(* Status Word *)
	stStatusData.bEnableOutputStage		:= fVelocity <> 0;
	stStatusData.bInverterReady   		:= TRUE;
	stStatusData.bPoDataEnable    		:= FALSE;
	stStatusData.bReserved3       		:= FALSE;
	stStatusData.bReserved4       		:= FALSE;
	stStatusData.bError           		:= FALSE;
	stStatusData.bReserved6       		:= FALSE;
	stStatusData.bReserved7       		:= FALSE;
	stStatusData.nStatus				:= 0;
END_METHOD

METHOD INTERNAL GetControlData
VAR_INPUT
	stControl 		: REFERENCE TO ST_SimMovitracControlData;
	pAddr			: ULINT; //PO adress
	bSwap 			: BOOL; //Swap BE_TO_HOST
END_VAR

VAR
	nCtrlIndex		: DWORD;
	nSpeedIndex		: DWORD;
	nRampIndex		: DWORD;
END_VAR
IF pAddr <= 0 THEN RETURN; END_IF

nCtrlIndex := stConfig.nCtrlAssign;
nSpeedIndex := stConfig.nSpeedAssign;
nRampIndex := stConfig.nRampAssign;

IF stConfig.bSwapProcessData THEN
	MEMCPY(ADR(stControlData) + 1, pAddr + nCtrlIndex, 1);
	MEMCPY(ADR(stControlData), pAddr + nCtrlIndex + 1, 1);
	MEMCPY(ADR(stControlData.nSetpointSpeed) + 1, pAddr + nSpeedIndex, 1);
	MEMCPY(ADR(stControlData.nSetpointSpeed), pAddr + nSpeedIndex + 1, 1);
ELSE
	MEMCPY(ADR(stControlData), pAddr + nCtrlIndex, 2);
	MEMCPY(ADR(stControlData.nSetpointSpeed), pAddr + nSpeedIndex, 2);
END_IF
END_METHOD

METHOD INTERNAL InitRun : BOOL
VAR_INST
	bInitRun : BOOL := TRUE;
END_VAR
IF NOT bInitRun THEN RETURN; END_IF
bInitRun := FALSE;

IF pControlData = 0 OR pStatusData = 0 THEN
	ADSLOGSTR(ADSLOG_MSGTYPE_WARN, CONCAT(sPath, ': %s'), 'Plc address not set.');
END_IF
END_METHOD

METHOD INTERNAL SetStatusData
VAR_INPUT
	stStatus 		: ST_SimMovitracStatusData;
	pAddr			: ULINT;
	bSwap 			: BOOL;
END_VAR

VAR
	nStatusIndex	: DWORD;
	nSpeedIndex	: DWORD;
END_VAR
IF pAddr <= 0 THEN RETURN; END_IF

nStatusIndex := stConfig.nStatusAssign;
nSpeedIndex := stConfig.nSpeedActAssign;

IF stConfig.bSwapProcessData THEN
	MEMCPY(pAddr + nStatusIndex + 1, ADR(stStatusData), 1);
	MEMCPY(pAddr + nStatusIndex, ADR(stStatusData.nStatus), 1);
	MEMCPY(pAddr + nSpeedIndex + 1, ADR(stStatusData.nActSpeed), 1);
	MEMCPY(pAddr + nSpeedIndex, ADR(stStatusData.nActSpeed) + 1, 1);	
ELSE
	MEMCPY(pAddr + nStatusIndex, ADR(stStatusData), 2);
	MEMCPY(pAddr + nSpeedIndex, ADR(stStatusData.nActSpeed), 2);
END_IF
END_METHOD

END_FUNCTION_BLOCK

// Devices/Drives/FB_SimMovitrac/FB_SimMovitracLTEB
FUNCTION_BLOCK FB_SimMovitracLTEB EXTENDS FB_LinkDataReal
VAR_INPUT
	bSTO					: BOOL := TRUE;
	bEnable 				: BOOL;
	bReverse				: BOOL;
	nTargetSpeed			: UINT; // Unit [INC]
	stConfig				: ST_SimMovitracConfig;
END_VAR

VAR_OUTPUT
	fActualSpeed			: REAL; // Units [RPM]
	bReady 					: BOOL;
	bRunning 				: BOOL;
END_VAR

VAR
	fAcc 					: REAL;
END_VAR

VAR CONSTANT
	
	MAX_VALUE_UINT 			: UINT := 65535; 
END_VAR

SUPER^();
InitRun();
ControlLogic();

METHOD PRIVATE ControlLogic
VAR
	fTargetSpeedInPercent	: REAL;
	fTargetSpeed 			: REAL;
END_VAR
// Start inverter 
IF bEnable AND bSTO THEN
	fTargetSpeedInPercent := F_Norm(0, MAX_VALUE_UINT, ABS(UINT_TO_REAL(nTargetSpeed))); // [INC] to [%] 
	fTargetSpeed := stConfig.fReferenceVelocity * fTargetSpeedInPercent; // [RPM]
	
	IF bReverse THEN
		ControlData := fTargetSpeed * -1;
	ELSE 
		ControlData := fTargetSpeed;
	END_IF
ELSE 
	ControlData := 0; 
END_IF

// Send values to the simulation interface
Control.0 := bEnable AND bSTO;

// Receive values from the simulation interface 
fActualSpeed := StatusData * stConfig.fGearFactor;
bReady  	 := NOT bEnable AND bSTO;
bRunning 	 := Status.0;
END_METHOD

METHOD PRIVATE InitRun
VAR_INST
	bInitRun : BOOL := TRUE;
END_VAR
IF NOT bInitRun THEN RETURN; END_IF
bInitRun := FALSE;

fAcc := stConfig.fReferenceVelocity * 1000 / stConfig.fProcessRamp;
END_METHOD

END_FUNCTION_BLOCK

// Devices/Drives/FB_Starter/FB_Starter
{attribute 'reflection'}
FUNCTION_BLOCK FB_Starter EXTENDS FB_LinkDataREAL
VAR_INPUT
	stControlData		: ST_StarterControlData;
	stConfig			: ST_StarterConfig;	
END_VAR

VAR_OUTPUT
	stStatusData		: ST_StarterStatusData;	
	fSpeed				: REAL; // Units [RPM]
END_VAR

VAR
	{attribute 'instance-path'}
	{attribute 'noinit'}
	sPath				: STRING;	
                    	
	fbDriveControl		: FB_DriveControl;
	bMoveActive			: BOOL;
	
	pControlData		: POINTER TO BYTE; //Addr. Process Output (PO), 2 BYTES FROM FIELDBUS
	pStatusData			: POINTER TO BYTE; //Addr. Process Input (PI), 2 BYTES FROM FIELDBUS
END_VAR

SUPER^();
InitRun();

GetControlData(stControlData, pControlData, stConfig.bSwapProcessData);
ControlLogic();
SetStatusData(stStatusData, pStatusData, stConfig.bSwapProcessData);

(*Assign Process Data Objects to device*)
METHOD PUBLIC AssignProcessData : BOOL
VAR_INPUT
	aControlData 		: ANY; //Addr. Process Output (PO), 2 BYTES FROM FIELDBUS
	aStatusData 		: ANY; //Addr. Process Input (PI), 2 BYTES TO FIELDBUS
END_VAR
THIS^.pControlData := aControlData.pValue;
THIS^.pStatusData := aStatusData.pValue;
END_METHOD

METHOD INTERNAL ControlLogic
(* Set parameter *)	
	bMoveActive := FALSE;
	
	IF (stControlData.MotorCW AND NOT stControlData.MotorCCW AND stControlData.BrakeActuation AND NOT stStatusData.GroupFault) THEN
		fbDriveControl.MoveVelocity(
			(stConfig.fVelocity),
			(stConfig.fAcceleration),
			(stConfig.fDeceleration));
		bMoveActive := TRUE;
	END_IF
	
	IF (stControlData.MotorCCW AND NOT stControlData.MotorCW AND stControlData.BrakeActuation AND NOT stStatusData.GroupFault) THEN
		fbDriveControl.MoveVelocity(
			(-stConfig.fVelocity),
			(stConfig.fAcceleration),
			(stConfig.fDeceleration));
		bMoveActive := TRUE;
	END_IF
	
	IF NOT bMoveActive OR stStatusData.GroupFault THEN
		fbDriveControl.Stop(stConfig.fDeceleration);
	END_IF

ControlData := fSpeed := fbDriveControl.fVelocity;
	
stStatusData.Ready 				:= TRUE;
stStatusData.MotorON 			:= NOT F_Compare(fbDriveControl.fVelocity, 0, 0.001); 
stStatusData.GroupFault 		:= FALSE;
stStatusData.GroupWarn 			:= FALSE;
stStatusData.Input1 			:= FALSE;
stStatusData.Input2 			:= FALSE;
stStatusData.Input3 			:= FALSE;
stStatusData.Input4 			:= FALSE;
stStatusData.MotorCurrent0 		:= FALSE;
stStatusData.MotorCurrent1 		:= FALSE;
stStatusData.MotorCurrent2 		:= FALSE;
stStatusData.MotorCurrent3 		:= FALSE;
stStatusData.MotorCurrent4 		:= FALSE;
stStatusData.MotorCurrent5 		:= FALSE;
stStatusData.ManualLocalMode	:= FALSE;
stStatusData.RampOperation 		:= FALSE;
END_METHOD

METHOD INTERNAL GetControlData
VAR_INPUT
	stControl 		: REFERENCE TO ST_StarterControlData;
	pAddr			: ULINT; //PO adress
	bSwap 			: BOOL; //Swap BE_TO_HOST
END_VAR

VAR	
	nControlWord 	: WORD;
END_VAR
IF pAddr <= 0 THEN RETURN; END_IF

IF bSwap THEN 
	MEMCPY(ADR(nControlWord), pAddr, 2);
	nControlWord := BE16_TO_HOST(nControlWord);
	MEMCPY(ADR(stControl), ADR(nControlWord), 2);
ELSE
	MEMCPY(ADR(stControl), pAddr, 2);
END_IF
END_METHOD

METHOD INTERNAL InitRun
VAR_INST
	bInitRun : BOOL := TRUE;
END_VAR
IF NOT bInitRun THEN RETURN; END_IF
bInitRun := FALSE;

IF pControlData = 0 OR pStatusData = 0 THEN
	ADSLOGSTR(ADSLOG_MSGTYPE_WARN, CONCAT(sPath, ': %s'), 'Plc address not set.');
END_IF

fbDriveControl.fPositionLimitMin := 0;
fbDriveControl.fPositionLimitMax := 0;
fbDriveControl.fAccMax := 0;
fbDriveControl.fTolerance := 0.1;
END_METHOD

METHOD INTERNAL SetStatusData
VAR_INPUT
	stStatus 		: ST_StarterStatusData;
	pAddr			: ULINT;
	bSwap 			: BOOL;
END_VAR

VAR
	nStatusWord 	: WORD;
END_VAR
IF pAddr <= 0 THEN RETURN; END_IF

IF bSwap THEN 
	MEMCPY(ADR(nStatusWord), ADR(stStatus), 2);
	nStatusWord := HOST_TO_BE16(nStatusWord);
	MEMCPY(pAddr, ADR(nStatusWord), 2);
ELSE
	MEMCPY(pAddr, ADR(stStatus), 2);
END_IF
END_METHOD

END_FUNCTION_BLOCK

// Devices/Safety/FB_EuchnerMGB
FUNCTION_BLOCK FB_EuchnerMGB EXTENDS FB_LinkDevice
VAR_INPUT
	bLock 					: BOOL; //Deactivates the tightening magnet
	bLockGuardMonitoring	: BOOL := TRUE; //Guard lock monitoring 0- 
	bReset 					: BOOL; //Error acknowledgement
	bLamp_1					: BOOL; //User defined input for item 1
	bLamp_2					: BOOL; //User defined input for item 2
	bLamp_3					: BOOL; //User defined input for item 3
	bLamp_4					: BOOL; //User defined input for item 4
END_VAR
VAR_OUTPUT
	bClosed 				: BOOL; //Door is closed
	bClosedAndLocked 		: BOOL; //Door is closed and guard locked / interlocked
	bButton_1				: BOOL; //User defined output for item 1
	bButton_2				: BOOL;	//User defined output for item 2
	bButton_3				: BOOL; //User defined output for item 3
	bButton_4				: BOOL; //User defined output for item 4
END_VAR

SUPER^();

Control.0 			:= bLock;
Control.1 			:= bReset;
Control.4 			:= bLamp_1;
Control.5 			:= bLamp_2;
Control.6 			:= bLamp_3;
Control.7 			:= bLamp_4;

bClosed 			:= Status.0;

IF bLockGuardMonitoring THEN
	bClosedAndLocked 	:= Status.1;
ELSE
	bClosedAndLocked 	:= Status.0;	
END_IF

bButton_1 			:= Status.4;
bButton_2 			:= Status.5;
bButton_3 			:= Status.6;
bButton_4 			:= Status.7;

END_FUNCTION_BLOCK

// Devices/Safety/FB_EuchnerSTP
FUNCTION_BLOCK FB_EuchnerSTP EXTENDS FB_LinkDevice
VAR_INPUT
	bLock 				: BOOL; //Deactivates the tightening magnet
	bLamp_RD			: BOOL; //User defined input for item 1
	bLamp_GN			: BOOL; //User defined input for item 2
END_VAR
VAR_OUTPUT
	bClosed 			: BOOL; //Door is closed
	bClosedAndLocked 	: BOOL; //Door is closed and guard locked / interlocked
END_VAR

SUPER^();
Control.0 			:= bLock;

Control.4 			:= bLamp_RD;
Control.5 			:= bLamp_GN;

bClosed 			:= Status.0;
bClosedAndLocked    := Status.1 OR (bLock AND bClosed);

END_FUNCTION_BLOCK

// Tests/Common/FB_AdsMessageHandler_Test
FUNCTION_BLOCK FB_AdsMessageHandler_Test EXTENDS TcUnit.FB_TestSuite
VAR
	stAdsMessageSend 		: ST_AdsMessage;
END_VAR

stAdsMessageSend.nIdxGrp := 16#80000005;
stAdsMessageSend.nIdxOffs := 7;
TestCaseWrite('ADS Write Indication 1', stAdsMessageSend);

stAdsMessageSend.nIdxGrp := 16#80000006;
stAdsMessageSend.nIdxOffs := 8;
TestCaseWrite('ADS Write Indication 2', stAdsMessageSend);

stAdsMessageSend.nIdxGrp := 16#80000007;
stAdsMessageSend.nIdxOffs := 9;
TestCaseWrite('ADS Write Indication 3', stAdsMessageSend);

stAdsMessageSend.nIdxGrp := 16#80000005;
stAdsMessageSend.nIdxOffs := 7;
TestCaseRead('ADS Read Indication 1', stAdsMessageSend);

stAdsMessageSend.nIdxGrp := 16#80000006;
stAdsMessageSend.nIdxOffs := 8;
TestCaseRead('ADS Read Indication 2', stAdsMessageSend);

stAdsMessageSend.nIdxGrp := 16#80000007;
stAdsMessageSend.nIdxOffs := 9;
TestCaseRead('ADS Read Indication 3', stAdsMessageSend);

METHOD TestCaseRead : REFERENCE TO FB_Test
VAR_INPUT
	sName 					: T_MaxString;
	stAdsMessage 			: ST_AdsMessage;
END_VAR

VAR
	fbAdsMessageHandler 	: FB_AdsMessageHandler;		
	fbAdsRead				: ADSREAD := (NETID := '', PORT := 851, TMOUT := DEFAULT_ADS_TIMEOUT);
	aData 					: ARRAY[0..5] OF BYTE;
	bResult 				: BOOL; 	
	stAdsMessageResult 	: ST_AdsMessage;
END_VAR
TEST(sName);

fbAdsRead(READ := FALSE);
fbAdsRead(IDXGRP := stAdsMessageSend.nIdxGrp, 
		IDXOFFS := stAdsMessageSend.nIdxOffs, 
        LEN := stAdsMessageSend.nLength, 
		DESTADDR := ADR(aData), 
        READ := TRUE);			

fbAdsMessageHandler.bVerbose := TRUE;			
fbAdsMessageHandler();

bResult := fbAdsMessageHandler.bIsAdsMessageReadValid;
stAdsMessageResult := fbAdsMessageHandler.stAdsMessageRead;

AssertTrue(bResult, 'Result value is not correct');

AssertEquals(Expected := stAdsMessage.tNetID,
Actual := stAdsMessageResult.tNetID,
Message := 'tNetID is not valid');

AssertEquals(Expected := stAdsMessage.nIdxGrp,
Actual := stAdsMessageResult.nIdxGrp,
Message := 'nIdxGrp is not valid');

AssertEquals(Expected := stAdsMessage.nIdxOffs,
Actual := stAdsMessageResult.nIdxOffs,
Message := 'nIdxOffs is not valid');

AssertEquals(Expected := stAdsMessage.nLength,
Actual := stAdsMessageResult.nLength,
Message := 'nLength is not valid');

TEST_FINISHED();
END_METHOD

METHOD TestCaseWrite : REFERENCE TO FB_Test
VAR_INPUT
	sName 					: T_MaxString;
	stAdsMessage 			: ST_AdsMessage;
END_VAR

VAR
	fbAdsMessageHandler 	: FB_AdsMessageHandler;		
	fbAdsWrite				: ADSWRITE := (NETID := '', PORT := 851, TMOUT := DEFAULT_ADS_TIMEOUT);
	aData 					: ARRAY[0..5] OF BYTE;
	bResult 				: BOOL; 	
	stAdsMessageResult 	: ST_AdsMessage;
END_VAR
TEST(sName);

fbAdsWrite(WRITE := FALSE);
fbAdsWrite(	IDXGRP := stAdsMessageSend.nIdxGrp, 
			IDXOFFS := stAdsMessageSend.nIdxOffs, 
            LEN := stAdsMessageSend.nLength, 
			SRCADDR := ADR(aData), 
            WRITE := TRUE);			

fbAdsMessageHandler.bVerbose := TRUE;			
fbAdsMessageHandler();

bResult := fbAdsMessageHandler.bIsAdsMessageWriteValid;
stAdsMessageResult := fbAdsMessageHandler.stAdsMessageWrite;

AssertTrue(bResult, 'Result value is not correct');

AssertEquals(Expected := stAdsMessage.tNetID,
Actual := stAdsMessageResult.tNetID,
Message := 'tNetID is not valid');

AssertEquals(Expected := stAdsMessage.nIdxGrp,
Actual := stAdsMessageResult.nIdxGrp,
Message := 'nIdxGrp is not valid');

AssertEquals(Expected := stAdsMessage.nIdxOffs,
Actual := stAdsMessageResult.nIdxOffs,
Message := 'nIdxOffs is not valid');

AssertEquals(Expected := stAdsMessage.nLength,
Actual := stAdsMessageResult.nLength,
Message := 'nLength is not valid');

TEST_FINISHED();
END_METHOD

END_FUNCTION_BLOCK

// Tests/Common/FB_Clamp01_Test
FUNCTION_BLOCK FB_Clamp01_Test EXTENDS TcUnit.FB_TestSuite

TestCase('Value Limit Min Overflow', fValue := -0.1, fExpected:= 0);
TestCase('Value Limit Min',fValue := 0.0, fExpected:= 0);
TestCase('Value In Range ',fValue := 0.5, fExpected:= 0.5);
TestCase('Value Limit Max',fValue := 1, fExpected:= 1);
TestCase('Value Limit Max Overflow',fValue := 1.1, fExpected:= 1);

METHOD TestCase
VAR_INPUT
	sName : T_MaxString;
	fValue : REAL;
	fExpected : REAL;
END_VAR

VAR	
	fResult : REAL;
END_VAR
TEST(sName);
	
fResult := F_Clamp01(fValue);
AssertEquals(Expected := fExpected,
             Actual := fResult,
             Message := 'Result value is not correct');	
	 
TEST_FINISHED();
END_METHOD

END_FUNCTION_BLOCK

// Tests/Common/FB_Compare_Test
FUNCTION_BLOCK FB_Compare_Test EXTENDS TcUnit.FB_TestSuite

TestCase('Compare Valid_1', fValueA := 0.0, fValueB := 0.0, fTolerance := 1E-6, bExpected:= TRUE);
TestCase('Compare Valid_2', fValueA := -1E-6, fValueB := -1E-6, fTolerance := 1E-6, bExpected:= TRUE);
TestCase('Compare Valid_3', fValueA := 1E-6, fValueB := 1E-6, fTolerance := 1E-6, bExpected:= TRUE);

TestCase('Compare Not Valid_1', fValueA := 0.0, fValueB := 0.00001, fTolerance := 1E-6, bExpected:= FALSE);
TestCase('Compare Not Valid_2', fValueA := -10, fValueB := -10.00001, fTolerance := 1E-6, bExpected:= FALSE);
TestCase('Compare Not Valid_3', fValueA := 100, fValueB := 100.00001, fTolerance := 1E-6, bExpected:= FALSE);

TestCase('Compare InRange_1', fValueA := 0.0, fValueB := 4.99999, fTolerance := 5, bExpected:= TRUE);
TestCase('Compare InRange_2', fValueA := -1, fValueB := -5.99999, fTolerance := 5, bExpected:= TRUE);
TestCase('Compare InRange_3', fValueA := 1, fValueB := 5.99999, fTolerance := 5, bExpected:= TRUE);

TestCase('Compare Not InRange_1', fValueA := 0.0, fValueB := 5.00000, fTolerance := 5, bExpected:= FALSE);
TestCase('Compare Not InRange_2', fValueA := -1, fValueB := -6.00000, fTolerance := 5, bExpected:= FALSE);
TestCase('Compare Not InRange_3', fValueA := 1, fValueB := 6.00000, fTolerance := 5, bExpected:= FALSE);

METHOD TestCase
VAR_INPUT
	sName : T_MaxString;
	fValueA : REAL;
	fValueB : REAL;
	fTolerance : REAL; 
	bExpected : BOOL;
END_VAR

VAR	
	bResult : BOOL;
END_VAR
TEST(sName);
	
bResult := F_Compare(fValueA, fValueB, fTolerance);
AssertEquals(Expected := bExpected,
             Actual := bResult,
             Message := 'Result value is not correct');	
	 
TEST_FINISHED();
END_METHOD

END_FUNCTION_BLOCK

// Tests/Common/FB_GetByte_Test
FUNCTION_BLOCK FB_GetByte_Test EXTENDS TcUnit.FB_TestSuite

TestGetLByte('Get LByte_1', nData := 16#1234, nExpected:= 16#34);
TestGetLByte('Get LByte_2', nData := 16#4321, nExpected:= 16#21);

TestGetHByte('Get HByte_1', nData := 16#1234, nExpected:= 16#12);
TestGetHByte('Get HByte_2', nData := 16#4321, nExpected:= 16#43);

METHOD TestGetHByte
VAR_INPUT
	sName : T_MaxString;	
	nData 	: WORD;
	nExpected : BYTE;
END_VAR

VAR		
	nResult : BYTE;
END_VAR
TEST(sName);


nResult := F_GetHByte(nData);
AssertEquals(Expected := nExpected,
             Actual := nResult,
             Message := 'Result value is not correct');	
	 
TEST_FINISHED();
END_METHOD

METHOD TestGetLByte
VAR_INPUT
	sName : T_MaxString;	
	nData 	: WORD;
	nExpected : BYTE;
END_VAR

VAR		
	nResult : BYTE;
END_VAR
TEST(sName);


nResult := F_GetLByte(nData);
AssertEquals(Expected := nExpected,
             Actual := nResult,
             Message := 'Result value is not correct');	
	 
TEST_FINISHED();
END_METHOD

END_FUNCTION_BLOCK

// Tests/Common/FB_InverBytesOrder_Test
FUNCTION_BLOCK FB_InverBytesOrder_Test EXTENDS TcUnit.FB_TestSuite

TestWord('Invert WORD_1', nData := 16#1234, nExpected:= 16#3412);
TestWord('Invert WORD_2', nData := 16#4321, nExpected:= 16#2143);

TestDWord('Invert DWORD_1', nData := 16#12345678, nExpected:= 16#78563412);
TestDWord('Invert DWORD_2', nData := 16#87654321, nExpected:= 16#21436587);

TestLWord('Invert LWORD_1', nData := 16#1234567812345678, nExpected:= 16#7856341278563412);
TestLWord('Invert LWORD_2', nData := 16#8765432187654321, nExpected:= 16#2143658721436587);

METHOD TestDWord
VAR_INPUT
	sName : T_MaxString;	
	nData 	: DWORD;
	nExpected : DWORD;
END_VAR

VAR		
	nResult : DWORD;
END_VAR
TEST(sName);


F_InverBytesOrder(nData);
AssertEquals(Expected := nExpected,
             Actual := nData,
             Message := 'Result value is not correct');	
	 
TEST_FINISHED();
END_METHOD

METHOD TestLWord
VAR_INPUT
	sName : T_MaxString;	
	nData 	: LWORD;
	nExpected : LWORD;
END_VAR

VAR		
	nResult : LWORD;
END_VAR
TEST(sName);


F_InverBytesOrder(nData);
AssertEquals(Expected := nExpected,
             Actual := nData,
             Message := 'Result value is not correct');	
	 
TEST_FINISHED();
END_METHOD

METHOD TestWord
VAR_INPUT
	sName : T_MaxString;	
	nData 	: WORD;
	nExpected : WORD;
END_VAR

VAR		
	nResult : WORD;
END_VAR
TEST(sName);


F_InverBytesOrder(nData);
AssertEquals(Expected := nExpected,
             Actual := nData,
             Message := 'Result value is not correct');	
	 
TEST_FINISHED();
END_METHOD

END_FUNCTION_BLOCK

// Tests/Common/FB_Norm_Test
FUNCTION_BLOCK FB_Norm_Test EXTENDS TcUnit.FB_TestSuite

TestCase('Normalize in Range_1', fMin := 0.0, fMax := 100, fValue := 0, fExpected:= 0);
TestCase('Normalize in Range_2', fMin := 0.0, fMax := 100, fValue := 20, fExpected:= 0.2);
TestCase('Normalize in Range_3', fMin := 0.0, fMax := 100, fValue := 70, fExpected:= 0.7);
TestCase('Normalize in Range_4', fMin := 0.0, fMax := 100, fValue := 100, fExpected:= 1);
TestCase('Normalize in Range_5', fMin := -100, fMax := 100, fValue := 0, fExpected:= 0.5);

TestCase('Normalize Overflow_1', fMin := -100, fMax := 100, fValue := -101, fExpected:= 0);
TestCase('Normalize Overflow_2', fMin := -100, fMax := 100, fValue := 101, fExpected:= 1);

METHOD TestCase
VAR_INPUT
	sName : T_MaxString;
	fMin : REAL;
	fMax : REAL;
	fValue : REAL; 
	fExpected : REAL;
END_VAR

VAR	
	fResult : REAL;
END_VAR
TEST(sName);
	
fResult := F_Norm(fMin, fMax, fValue);
AssertEquals(Expected := fExpected,
             Actual := fResult,
             Message := 'Result value is not correct');	
	 
TEST_FINISHED();
END_METHOD

END_FUNCTION_BLOCK

// Tests/Common/FB_RecordData_Test
FUNCTION_BLOCK FB_RecordData_Test EXTENDS TcUnit.FB_TestSuite
VAR
	fbAdsMessageHandler 	: FB_AdsMessageHandler;
	fbRecordData 			: FB_RecordData(refAdsMessageHandler := fbAdsMessageHandler);	
	
	stAdsHandlerMessage 	: ST_AdsMessage;
	stDeviceMessage 		: ST_AdsMessage;
END_VAR

TestCasesCompare();
TestGetReadIndication();
TestGetWriteIndication();
TestSendReadResponse();
TestSendWriteResponse();
TestAutoResponseWriteMessage();
TestAutoResponseReadMessage();

METHOD TestAutoResponseReadMessage : REFERENCE TO FB_Test
VAR
	fbAdsRead				: ADSREAD := (NETID := '', PORT := 851, TMOUT := DEFAULT_ADS_TIMEOUT);
	stAdsMessage			: REFERENCE TO ST_AdsMessage;
	nData					: BYTE;
	bResult 				: BOOL;
	bResultPort 			: T_AmsPort;
	nExpectedPort			: T_AmsPort;
END_VAR
TEST('Auto Response Ads Read Message');

stAdsHandlerMessage.tPort := 351; 
stAdsHandlerMessage.nInvokeID := 500;
stAdsHandlerMessage.nIdxGrp := 16#80000001;
stAdsHandlerMessage.nIdxOffs := 10;
stDeviceMessage.tPort := 351;
stDeviceMessage.nInvokeID := 500;
stDeviceMessage.nIdxGrp := 16#80000001;
stDeviceMessage.nIdxOffs := 10;

fbAdsRead(READ := FALSE);
fbAdsRead(	IDXGRP := stAdsHandlerMessage.nIdxGrp, 
			IDXOFFS := stAdsHandlerMessage.nIdxOffs, 
        	LEN := stAdsHandlerMessage.nLength, 
			DESTADDR := ADR(nData), 
        	READ := TRUE);			

fbAdsMessageHandler.bLog := TRUE;
fbAdsMessageHandler.bVerbose := TRUE;	
fbRecordData.eControllerType := E_ControllerType.PlcSimAdvanced;

fbRecordData();		
fbAdsMessageHandler();

bResult := fbAdsMessageHandler.bIsAdsMessageReadValid;
AssertTrue(bResult, 'AdsMessageReadValid expected TRUE');

fbRecordData();	
fbAdsMessageHandler();
bResult := fbAdsMessageHandler.bIsAdsMessageReadValid;
AssertFalse(bResult, 'AdsMessageReadValid expected FALSE');

nExpectedPort := 0;
bResultPort := fbAdsMessageHandler.stAdsMessageRead.tPort;

AssertEquals(Expected := nExpectedPort,
	Actual := bResultPort,
	Message := 'tPort value is incorrect');

TEST_FINISHED();
END_METHOD

METHOD TestAutoResponseWriteMessage : REFERENCE TO FB_Test
VAR
	fbAdsWrite				: ADSWRITE := (NETID := '', PORT := 851, TMOUT := DEFAULT_ADS_TIMEOUT);
	stAdsMessage			: REFERENCE TO ST_AdsMessage;
	nData					: BYTE;
	bResult 				: BOOL;
	bResultPort 			: T_AmsPort;
	nExpectedPort			: T_AmsPort;
END_VAR
TEST('Auto Response Ads Write Message');

stAdsHandlerMessage.tPort := 351; 
stAdsHandlerMessage.nInvokeID := 500;
stAdsHandlerMessage.nIdxGrp := 16#80000001;
stAdsHandlerMessage.nIdxOffs := 10;
stDeviceMessage.tPort := 351;
stDeviceMessage.nInvokeID := 500;
stDeviceMessage.nIdxGrp := 16#80000001;
stDeviceMessage.nIdxOffs := 10;

fbAdsWrite(WRITE := FALSE);
fbAdsWrite(	IDXGRP := stAdsHandlerMessage.nIdxGrp, 
			IDXOFFS := stAdsHandlerMessage.nIdxOffs, 
           	LEN := stAdsHandlerMessage.nLength, 
			SRCADDR := ADR(nData), 
           	WRITE := TRUE);			

fbAdsMessageHandler.bLog := TRUE;
fbAdsMessageHandler.bVerbose := TRUE;	
fbRecordData.eControllerType := E_ControllerType.PlcSimAdvanced;

fbRecordData();		
fbAdsMessageHandler();

bResult := fbAdsMessageHandler.bIsAdsMessageWriteValid;
AssertTrue(bResult, 'AdsMessageWriteValid expected TRUE');

fbRecordData();	
fbAdsMessageHandler();
bResult := fbAdsMessageHandler.bIsAdsMessageWriteValid;
AssertFalse(bResult, 'AdsMessageWriteValid expected FALSE');

nExpectedPort := 0;
bResultPort := fbAdsMessageHandler.stAdsMessageWrite.tPort;

AssertEquals(Expected := nExpectedPort,
	Actual := bResultPort,
	Message := 'tPort value is incorrect');

TEST_FINISHED();
END_METHOD

METHOD TestCaseCompare : REFERENCE TO FB_Test
VAR_INPUT
	sName 					: T_MaxString;
	stAdsHandlerMessage 	: ST_AdsMessage;
	stDeviceMessage 		: ST_AdsMessage;
	bExpected				: BOOL;
END_VAR

VAR
	bResult 				: BOOL;
END_VAR
TEST(sName);

bResult := fbRecordData.DataValid(stDeviceMessage, stAdsHandlerMessage);

AssertEquals(Expected := bExpected,
	Actual := bResult,
	Message := 'Expected compare result is wrong');

IF bResult AND bExpected THEN
	bResult := stAdsHandlerMessage.tPort = 0;
	AssertTrue(bResult, 'tPort must be 0');
END_IF
	
	
TEST_FINISHED();
END_METHOD

ACTION TestCasesCompare:
(*Test ADS Message compare*)
stAdsHandlerMessage.tPort := 351; 
stAdsHandlerMessage.nInvokeID := 500;
stAdsHandlerMessage.nIdxGrp := 16#80000001;
stAdsHandlerMessage.nIdxOffs := 10;
stDeviceMessage.tPort := 351;
stDeviceMessage.nInvokeID := 500;
stDeviceMessage.nIdxGrp := 16#80000001;
stDeviceMessage.nIdxOffs := 10;
TestCaseCompare('Compare TRUE 1', stAdsHandlerMessage, stDeviceMessage, TRUE);

stAdsHandlerMessage.tPort := 351; 
stAdsHandlerMessage.nInvokeID := 16#12340011;
stAdsHandlerMessage.nIdxGrp := 16#80000001;
stAdsHandlerMessage.nIdxOffs := 10;
stDeviceMessage.tPort := 351;
stDeviceMessage.nInvokeID := 16#43210011;
stDeviceMessage.nIdxGrp := 16#80000001;
stDeviceMessage.nIdxOffs := 10;
TestCaseCompare('Compare TRUE - InvokeID', stAdsHandlerMessage, stDeviceMessage, TRUE);

stAdsHandlerMessage.tPort := 351; 
stAdsHandlerMessage.nInvokeID := 16#12340011;
stAdsHandlerMessage.nIdxGrp := 16#80000001;
stAdsHandlerMessage.nIdxOffs := 10;
stDeviceMessage.tPort := 351;
stDeviceMessage.nInvokeID := 16#43210011;
stDeviceMessage.nIdxGrp := 16#80000001;
stDeviceMessage.nIdxOffs := 10;
TestCaseCompare('Compare TRUE - nIdxOffs', stAdsHandlerMessage, stDeviceMessage, TRUE);

stAdsHandlerMessage.tPort := 351; 
stAdsHandlerMessage.nInvokeID := 16#12340011;
stAdsHandlerMessage.nIdxGrp := 16#80000001;
stAdsHandlerMessage.nIdxOffs := 10;
stDeviceMessage.tPort := 351;
stDeviceMessage.nInvokeID := 16#43210011;
stDeviceMessage.nIdxGrp := 16#80000001;
stDeviceMessage.nIdxOffs := 16#FFFFFFFF;
TestCaseCompare('Compare TRUE - nIdxOffs 16#FFFFFFFF', stAdsHandlerMessage, stDeviceMessage, TRUE);

stAdsHandlerMessage.tPort := 351; 
stAdsHandlerMessage.nInvokeID := 16#12340011;
stAdsHandlerMessage.nIdxGrp := 16#12340011;
stAdsHandlerMessage.nIdxOffs := 10;
stDeviceMessage.tPort := 351;
stDeviceMessage.nInvokeID := 16#43210011;
stDeviceMessage.nIdxGrp := 16#43210011;
stDeviceMessage.nIdxOffs := 10;
TestCaseCompare('Compare TRUE - nIdxGrp', stAdsHandlerMessage, stDeviceMessage, TRUE);

stAdsHandlerMessage.tPort := 351; 
stAdsHandlerMessage.nInvokeID := 16#12340011;
stAdsHandlerMessage.nIdxGrp := 16#12340011;
stAdsHandlerMessage.nIdxOffs := 10;
stDeviceMessage.tPort := 351;
stDeviceMessage.nInvokeID := 16#43210011;
stDeviceMessage.nIdxGrp := 0;
stDeviceMessage.nIdxOffs := 10;
TestCaseCompare('Compare TRUE - nIdxGrp 0', stAdsHandlerMessage, stDeviceMessage, TRUE);

stAdsHandlerMessage.tPort := 0; 
stAdsHandlerMessage.nInvokeID := 500;
stAdsHandlerMessage.nIdxGrp := 16#80000001;
stAdsHandlerMessage.nIdxOffs := 10;
stDeviceMessage.tPort := 351;
stDeviceMessage.nInvokeID := 500;
stDeviceMessage.nIdxGrp := 16#80000001;
stDeviceMessage.nIdxOffs := 10;
TestCaseCompare('Compare FALSE - AdsHandler Port 0', stAdsHandlerMessage, stDeviceMessage, FALSE);

stAdsHandlerMessage.tPort := 351; 
stAdsHandlerMessage.nInvokeID := 16#12340010;
stAdsHandlerMessage.nIdxGrp := 16#80000001;
stAdsHandlerMessage.nIdxOffs := 10;
stDeviceMessage.tPort := 351;
stDeviceMessage.nInvokeID := 16#43210001;
stDeviceMessage.nIdxGrp := 16#80000001;
stDeviceMessage.nIdxOffs := 10;
TestCaseCompare('Compare FALSE - InvokeID', stAdsHandlerMessage, stDeviceMessage, FALSE);

stAdsHandlerMessage.tPort := 351; 
stAdsHandlerMessage.nInvokeID := 16#12340011;
stAdsHandlerMessage.nIdxGrp := 16#12340000;
stAdsHandlerMessage.nIdxOffs := 10;
stDeviceMessage.tPort := 351;
stDeviceMessage.nInvokeID := 16#43210000;
stDeviceMessage.nIdxGrp := 16#43210022;
stDeviceMessage.nIdxOffs := 10;
TestCaseCompare('Compare FALSE - nIdxGrp', stAdsHandlerMessage, stDeviceMessage, FALSE);

stAdsHandlerMessage.tPort := 351; 
stAdsHandlerMessage.nInvokeID := 16#12340011;
stAdsHandlerMessage.nIdxGrp := 16#12340000;
stAdsHandlerMessage.nIdxOffs := 20;
stDeviceMessage.tPort := 351;
stDeviceMessage.nInvokeID := 16#43210000;
stDeviceMessage.nIdxGrp := 16#43210000;
stDeviceMessage.nIdxOffs := 10;
TestCaseCompare('Compare FALSE - nIdxOffs', stAdsHandlerMessage, stDeviceMessage, FALSE);
END_ACTION

METHOD TestGetReadIndication : REFERENCE TO FB_Test
VAR	
	fbAdsRead				: ADSREAD := (NETID := '', PORT := 851, TMOUT := DEFAULT_ADS_TIMEOUT);
	stAdsMessage			: REFERENCE TO ST_AdsMessage;
	nData					: BYTE;
	bResult 				: BOOL;
END_VAR
TEST('Get Read Indication');

stAdsHandlerMessage.tPort := 351; 
stAdsHandlerMessage.nInvokeID := 500;
stAdsHandlerMessage.nIdxGrp := 16#80000001;
stAdsHandlerMessage.nIdxOffs := 10;
stDeviceMessage.tPort := 351;
stDeviceMessage.nInvokeID := 500;
stDeviceMessage.nIdxGrp := 16#80000001;
stDeviceMessage.nIdxOffs := 10;

fbAdsRead(READ := FALSE);
fbAdsRead(	IDXGRP := stAdsHandlerMessage.nIdxGrp, 
			IDXOFFS := stAdsHandlerMessage.nIdxOffs, 
        	LEN := stAdsHandlerMessage.nLength, 
			DESTADDR := ADR(nData), 
        	READ := TRUE);			

fbAdsMessageHandler.bLog := TRUE;
fbAdsMessageHandler.bVerbose := TRUE;			
fbAdsMessageHandler();

fbRecordData.eControllerType := E_ControllerType.PlcSimAdvanced;

bResult := fbRecordData.GetReadIndication(stDeviceMessage);
stAdsMessage REF= fbAdsMessageHandler.stAdsMessageRead;

AssertTrue(bResult, 'Result value is not correct');

bResult := stAdsMessage.tPort = 0;
AssertTrue(bResult, 'tPort must be 0');

TEST_FINISHED();
END_METHOD

METHOD TestGetWriteIndication : REFERENCE TO FB_Test
VAR	
	fbAdsWrite				: ADSWRITE := (NETID := '', PORT := 851, TMOUT := DEFAULT_ADS_TIMEOUT);
	stAdsMessage			: REFERENCE TO ST_AdsMessage;
	nData					: BYTE;
	bResult 				: BOOL;
END_VAR
TEST('Get Write Indication');

stAdsHandlerMessage.tPort := 351; 
stAdsHandlerMessage.nInvokeID := 500;
stAdsHandlerMessage.nIdxGrp := 16#80000001;
stAdsHandlerMessage.nIdxOffs := 10;
stDeviceMessage.tPort := 351;
stDeviceMessage.nInvokeID := 500;
stDeviceMessage.nIdxGrp := 16#80000001;
stDeviceMessage.nIdxOffs := 10;

fbAdsWrite(WRITE := FALSE);
fbAdsWrite(	IDXGRP := stAdsHandlerMessage.nIdxGrp, 
			IDXOFFS := stAdsHandlerMessage.nIdxOffs, 
           	LEN := stAdsHandlerMessage.nLength, 
			SRCADDR := ADR(nData), 
           	WRITE := TRUE);			

fbAdsMessageHandler.bLog := TRUE;
fbAdsMessageHandler.bVerbose := TRUE;			
fbAdsMessageHandler();

fbRecordData.eControllerType := E_ControllerType.PlcSimAdvanced;

bResult := fbRecordData.GetWriteIndication(stDeviceMessage);
stAdsMessage REF= fbAdsMessageHandler.stAdsMessageRead;

AssertTrue(bResult, 'Result value is not correct');

bResult := stAdsMessage.tPort = 0;
AssertTrue(bResult, 'tPort must be 0');

TEST_FINISHED();
END_METHOD

METHOD TestSendReadResponse : REFERENCE TO FB_Test
VAR
	stAdsMessage : ST_AdsMessage;
	hExpected : HRESULT;
	hRes : HRESULT;
END_VAR
TEST('Send Read Response');

stAdsMessage.tPort := 351;
stAdsMessage.nInvokeID := 500;
stAdsMessage.nIdxGrp := 16#80000001;
stAdsMessage.nIdxOffs := 10;

fbAdsMessageHandler.bLog := TRUE;
fbAdsMessageHandler.bVerbose := TRUE;			
fbAdsMessageHandler();

fbRecordData.eControllerType := E_ControllerType.PlcSimAdvanced;

hExpected := S_OK;
hRes := fbRecordData.SendReadResponse(stAdsMessage);

AssertEquals(Expected := hExpected,
	Actual := hRes,
	Message := 'Expected result is not valid');
	
TEST_FINISHED();
END_METHOD

METHOD TestSendWriteResponse : REFERENCE TO FB_Test
VAR
	stAdsMessage : ST_AdsMessage;
	hExpected : HRESULT;
	hRes : HRESULT;
END_VAR
TEST('Send Write Response');

stAdsMessage.tPort := 351;
stAdsMessage.nInvokeID := 500;
stAdsMessage.nIdxGrp := 16#80000001;
stAdsMessage.nIdxOffs := 10;

fbAdsMessageHandler.bLog := TRUE;
fbAdsMessageHandler.bVerbose := TRUE;			
fbAdsMessageHandler();

fbRecordData.eControllerType := E_ControllerType.PlcSimAdvanced;

hExpected := S_OK;
hRes := fbRecordData.SendReadResponse(stAdsMessage);

AssertEquals(Expected := hExpected,
	Actual := hRes,
	Message := 'Expected result is not valid');
	
TEST_FINISHED();
END_METHOD

END_FUNCTION_BLOCK

// Tests/Common/FB_Scale_Test
FUNCTION_BLOCK FB_Scale_Test EXTENDS TcUnit.FB_TestSuite

TestCase('Scale InRange_1', 
fInputMin := 0.0, fInputMax := 100, 
fOutputMin := 0, fOutputMax:= 1000, 
fValue := 0, fExpected:= 0);

TestCase('Scale InRange_2', 
fInputMin := 0.0, fInputMax := 100, 
fOutputMin := 0, fOutputMax:= 1000, 
fValue := 50, fExpected:= 500);

TestCase('Scale InRange_3', 
fInputMin := 0.0, fInputMax := 100, 
fOutputMin := 0, fOutputMax:= 1000, 
fValue := 100, fExpected:= 1000);

TestCase('Scale Overflow_1', 
fInputMin := 0.0, fInputMax := 100, 
fOutputMin := 0, fOutputMax:= 1000, 
fValue := -100, fExpected:= 0);

TestCase('Scale Overflow_2', 
fInputMin := 0.0, fInputMax := 100, 
fOutputMin := 0, fOutputMax:= 1000, 
fValue := 200, fExpected:= 1000);

TestInputValidation('Inputs Valid_1', 
fInputMin := 0.0, fInputMax := 100, 
fOutputMin := 0, fOutputMax:= 1000, bExpected:= FALSE);

TestInputValidation('Inputs Valid_2', 
fInputMin := 99.99, fInputMax := 100, 
fOutputMin := 999.99, fOutputMax:= 1000, bExpected:= FALSE);

TestInputValidation('Inputs Not Valid_1', 
fInputMin := 100, fInputMax := 100, 
fOutputMin := 0, fOutputMax:= 1000, bExpected:= TRUE);

TestInputValidation('Inputs Not Valid_2', 
fInputMin := 100.0001, fInputMax := 100, 
fOutputMin := 0, fOutputMax:= 1000, bExpected:= TRUE);

TestInputValidation('Inputs Not Valid_3', 
fInputMin := 0, fInputMax := 100, 
fOutputMin := 1000, fOutputMax:= 1000, bExpected:= TRUE);

TestInputValidation('Inputs Not Valid_4', 
fInputMin := 0, fInputMax := 100, 
fOutputMin := 1000.001, fOutputMax:= 1000, bExpected:= TRUE);

METHOD TestCase
VAR_INPUT
	sName : T_MaxString;	
	fInputMin 	: LREAL;
	fInputMax 	: LREAL;
	fOutputMin 	: LREAL;
	fOutputMax 	: LREAL;
	fValue 		: LREAL; 
	fExpected 	: LREAL;
END_VAR

VAR	
	fResult 	: LREAL;
END_VAR
TEST(sName);
	
fResult := F_ScaleLREAL(fValue, fInputMin, fInputMax, fOutputMin, fOutputMax);
AssertEquals(Expected := fExpected,
             Actual := fResult,
             Message := 'Result value is not correct');	
	 
TEST_FINISHED();
END_METHOD

METHOD TestInputValidation : REFERENCE TO FB_Test
VAR_INPUT
	sName : T_MaxString;	
	fInputMin 	: LREAL;
	fInputMax 	: LREAL;
	fOutputMin 	: LREAL;
	fOutputMax 	: LREAL;
	bExpected 	: BOOL;
END_VAR

VAR	
	bResult 	: BOOL;
END_VAR
TEST(sName);
	
F_ScaleLREAL(0, fInputMin, fInputMax, fOutputMin, fOutputMax, bError => bResult);
AssertEquals(Expected := bExpected,
             Actual := bResult,
             Message := 'Result value is not correct');	
	 
TEST_FINISHED();
END_METHOD

END_FUNCTION_BLOCK

// Tests/Common/FB_Sign_Test
FUNCTION_BLOCK FB_Sign_Test EXTENDS TcUnit.FB_TestSuite

TestCase('Sign Negative_1', fValue := -0.00001, fExpected:= -1);
TestCase('Sign Negative_2', fValue := -0.1, fExpected:= -1);
TestCase('Sign Negative_3', fValue := -1, fExpected:= -1);

TestCase('Sign Positive_1', fValue := 0, fExpected:= 1);
TestCase('Sign Positive_2', fValue := 0.00001, fExpected:= 1);
TestCase('Sign Positive_3', fValue := 0.1, fExpected:= 1);
TestCase('Sign Positive_4', fValue := 1, fExpected:= 1);

METHOD TestCase
VAR_INPUT
	sName : T_MaxString;	
	fValue : REAL; 
	fExpected : REAL;
END_VAR

VAR	
	fResult : REAL;
END_VAR
TEST(sName);
	
fResult := F_Sign(fValue);
AssertEquals(Expected := fExpected,
             Actual := fResult,
             Message := 'Result value is not correct');	
	 
TEST_FINISHED();
END_METHOD

END_FUNCTION_BLOCK

// Tests/Common/FB_System_Test
FUNCTION_BLOCK FB_System_Test EXTENDS TcUnit.FB_TestSuite
VAR
	fbSystem : FB_System;
END_VAR

TestInitialization();
TestProperties();

METHOD TestInitialization
VAR
	fbGetCurTaskIdx 	: TC2_SYSTEM.GETCURTASKINDEX;
	fResult 	: REAL;
	fExpected 	: REAL;
	bResult 	: BOOL;
	bExpected 	: BOOL;
END_VAR
TEST('Before InitRun fTimeScaling is 0');
fExpected := 0;
fResult := fbSystem.fTimeScaling;
AssertEquals(Expected := fExpected,
             Actual := fResult,
             Message := 'Result value is not correct');
TEST_FINISHED();

TEST('Before InitRun fDeltaTime is 0');
fExpected := 0;
fResult := fbSystem.fDeltaTime;
AssertEquals(Expected := fExpected,
             Actual := fResult,
             Message := 'Result value is not correct');	
TEST_FINISHED();

TEST('Before InitRun GVL_IOSEF.refSystem is NULL');
bExpected := FALSE;
bResult := __ISVALIDREF(GVL_Core.refSystem);
AssertEquals(Expected := bExpected,
             Actual := bResult,
             Message := 'Result value is not correct');	
TEST_FINISHED();

fbSystem();

TEST('After InitRun fTimeScaling > 0');
fExpected := 1;
fResult := fbSystem.fTimeScaling;
AssertEquals(Expected := fExpected,
             Actual := fResult,
             Message := 'Result value is not correct');
TEST_FINISHED();

TEST('After InitRun fDeltaTime > 0');
fbGetCurTaskIdx();
fExpected := UDINT_TO_REAL(TwinCAT_SystemInfoVarList._TaskInfo[fbGetCurTaskIdx.index].CycleTime / 10000) / 1000.0;
fResult := fbSystem.fDeltaTime;
AssertEquals(Expected := fExpected,
             Actual := fResult,
             Message := 'Result value is not correct');	
TEST_FINISHED();

TEST('After InitRun GVL_IOSEF.refSystem is Valid');
bExpected := TRUE;
bResult := __ISVALIDREF(GVL_Core.refSystem);
AssertEquals(Expected := bExpected,
             Actual := bResult,
             Message := 'Result value is not correct');	
TEST_FINISHED();
END_METHOD

METHOD TestProperties : REFERENCE TO FB_Test
VAR
	fbGetCurTaskIdx 	: TC2_SYSTEM.GETCURTASKINDEX;
	fResult 	: REAL;
	fExpected 	: REAL;
END_VAR
TEST('Test Property: bDebug');
fbSystem.bDebug := TRUE;
AssertTRUE(Condition := fbSystem.bDebug,  Message := 'Property value is not correct');	
TEST_FINISHED();

TEST('Test Property: bVerbose');
fbSystem.bVerbose := TRUE;
AssertTRUE(Condition := fbSystem.bVerbose,  Message := 'Property value is not correct');	
TEST_FINISHED();

TEST('Test Property: fTimeScaling Initial');
fExpected := 1;
fResult := fbSystem.fTimeScaling;
AssertEquals(Expected := fExpected,
             Actual := fResult,
             Message := 'Result value is not correct');
TEST_FINISHED();

TEST('Test Property: fTimeScaling Zero');
fbSystem.fTimeScaling := 0;
fExpected := 1;
fResult := fbSystem.fTimeScaling;
AssertEquals(Expected := fExpected,
             Actual := fResult,
             Message := 'Result value is not correct');
TEST_FINISHED();

TEST('Test Property: fTimeScaling Limit Min');
fbSystem.fTimeScaling := -1;
fExpected := 0.01000001;
fResult := fbSystem.fTimeScaling;
AssertEquals(Expected := fExpected,
             Actual := fResult,
             Message := 'Result value is not correct');
TEST_FINISHED();

TEST('Test Property: fTimeScaling Limit Max');
fbSystem.fTimeScaling := 1E+6;
fExpected := 100;
fResult := fbSystem.fTimeScaling;
AssertEquals(Expected := fExpected,
             Actual := fResult,
             Message := 'Result value is not correct');
TEST_FINISHED();

TEST('Test Property: fTimeScaling In Range_1');
fbSystem.fTimeScaling := 2;
fExpected := 2;
fResult := fbSystem.fTimeScaling;
AssertEquals(Expected := fExpected,
             Actual := fResult,
             Message := 'Result value is not correct');
TEST_FINISHED();

TEST('Test Property: fTimeScaling In Range_2');
fbSystem.fTimeScaling := 1;
fExpected := 1;
fResult := fbSystem.fTimeScaling;
AssertEquals(Expected := fExpected,
             Actual := fResult,
             Message := 'Result value is not correct');
TEST_FINISHED();
END_METHOD

END_FUNCTION_BLOCK

// Tests/Components/FB_DriveControl_Test
FUNCTION_BLOCK FB_DriveControl_Test EXTENDS TcUnit.FB_TestSuite

TestCaseMoveVelocityLimits();
TestProperties();

TestCaseMoveVelocity('Velocity Zero', 0, 0, TRUE);

TestCaseMoveVelocity('Target Positiv Velocity_1', 0, 10, TRUE);
TestCaseMoveVelocity('Target Positiv Velocity_2', 90, 100, TRUE);
TestCaseMoveVelocity('Target Positiv Velocity_3', 990, 1000, TRUE);
TestCaseMoveVelocity('Target Positiv Velocity_4', 50, 100, FALSE);
TestCaseMoveVelocity('Target Positiv Velocity_5', 500, 1000, FALSE);

TestCaseMoveVelocity('Target Negative Velocity_1', 0, -10, TRUE);
TestCaseMoveVelocity('Target Negative Velocity_2', -90, -100, TRUE);
TestCaseMoveVelocity('Target Negative Velocity_3', -990, -1000, TRUE);
TestCaseMoveVelocity('Target Negative Velocity_4', -50, -100, FALSE);
TestCaseMoveVelocity('Target Negative Velocity_5', -500, -1000, FALSE);

TestCaseMoveAbsolute('Move Positive Absolute_1', 0, 1, 1000, TRUE);
TestCaseMoveAbsolute('Move Positive Absolute_2', 0, 10, 1000, TRUE);
TestCaseMoveAbsolute('Move Positive Absolute_3', 0, 100, 1000, FALSE);
TestCaseMoveAbsolute('Move Positive Absolute_4', 0, 1000, 1000, FALSE);

TestCaseMoveAbsolute('Move Positive Absolute_11', 50, 51, 1000, TRUE);
TestCaseMoveAbsolute('Move Positive Absolute_12', 50, 60, 1000, TRUE);
TestCaseMoveAbsolute('Move Positive Absolute_13', -50, -49, 1000, TRUE);
TestCaseMoveAbsolute('Move Positive Absolute_14', -50, -40, 1000, TRUE);

TestCaseMoveAbsolute('Move Negative Absolute_1', 0, -1, 1000, TRUE);
TestCaseMoveAbsolute('Move Negative Absolute_2', 0, -10, 1000, TRUE);
TestCaseMoveAbsolute('Move Negative Absolute_3', 0, -100, 1000, FALSE);
TestCaseMoveAbsolute('Move Negative Absolute_4', 0, -1000, 1000, FALSE);

TestCaseMoveAbsolute('Move Negative Absolute_11', -50, -51, 1000, TRUE);
TestCaseMoveAbsolute('Move Negative Absolute_12', -50, -60, 1000, TRUE);
TestCaseMoveAbsolute('Move Negative Absolute_13', 50, 49, 1000, TRUE);
TestCaseMoveAbsolute('Move Negative Absolute_14', 50, 40, 1000, TRUE);

TestStop();

METHOD TestCaseMoveAbsolute
VAR_INPUT
	sName 				: T_MaxString;
	fInitPosition 		: REAL;
	fTargetPosition 	: REAL;
	fTargetVelocity 	: REAL;
	bExpected 			: BOOL;
END_VAR

VAR
	fbDriveControl 		: FB_DriveControl;
	nCycleCount 		: INT;
	bResult 			: BOOL;
	fResult 			: REAL;
	fVel 				: REAL;
	fExpectedVel 		: REAL := 0;
END_VAR
TEST(sName);

fbDriveControl.fPosition := fInitPosition;

FOR nCycleCount := 0 TO 10 DO
    fbDriveControl.MoveAbsolute(fTargetPosition, fTargetVelocity, 1E+6, 1E+6);
END_FOR

bResult := fbDriveControl.bIsPositionReached;
fResult := fbDriveControl.fPosition;
fVel := fbDriveControl.fVelocity;

AssertEquals(Expected := bExpected,
             Actual := bResult,
             Message := 'Position is not reached');

IF bExpected THEN
	AssertEquals(Expected := fTargetPosition,
             Actual := fResult,
             Message := 'Position value is not correct');	
	AssertEquals(Expected := fExpectedVel,
             Actual := fVel,
             Message := 'Velocity value is not correct');	
END_IF
	 
TEST_FINISHED();
END_METHOD

METHOD TestCaseMoveVelocity
VAR_INPUT
	sName 				: T_MaxString;
	fInitVelocity 		: REAL;
	fTargetVelocity 	: REAL;
	bExpected 			: BOOL;
END_VAR

VAR
	fbDriveControl 		: FB_DriveControl;
	nCycleCount 		: INT;
	bResult 			: BOOL;	
	fResult 			: REAL;	
END_VAR
TEST(sName);

fbDriveControl.fVelocity := fInitVelocity;

FOR nCycleCount := 0 TO 10 DO
    fbDriveControl.MoveVelocity(fTargetVelocity, 1000, 1000);
END_FOR;

fResult := fbDriveControl.fVelocity;

IF bExpected THEN
	AssertEquals(Expected := fTargetVelocity,
             Actual := fResult,
             Message := 'Velocity value is not correct');
ELSE
	bResult := F_Compare(fbDriveControl.fVelocity, fTargetVelocity, 1E-6);
	AssertFALSE(bResult, 'Not Expected Velocity');	 	
END_IF

TEST_FINISHED();
END_METHOD

METHOD TestCaseMoveVelocityLimits
VAR
	fbDriveControl 		: FB_DriveControl;
	nCycleCount 		: INT;
	bResult 			: BOOL;	
	fResult 			: REAL;	
	fExpected 			: REAL;
END_VAR
TEST('Position Limit Min');

fExpected := 0;
fbDriveControl.fPositionLimitMin := -10;
fbDriveControl.fPosition := -10;

fbDriveControl.MoveVelocity(1000, 1000, 1000);
fResult := fbDriveControl.fVelocity;

AssertEquals(Expected := fExpected,
             Actual := fResult,
             Message := 'Velocity value is not limited');

TEST_FINISHED();

TEST('Position Limit Max');

fExpected := 0;
fbDriveControl.fPositionLimitMax := 10;
fbDriveControl.fPosition := 10;

fbDriveControl.MoveVelocity(1000, 1000, 1000);
fResult := fbDriveControl.fVelocity;

AssertEquals(Expected := fExpected,
             Actual := fResult,
             Message := 'Velocity value is not limited');

TEST_FINISHED();
END_METHOD

METHOD TestProperties
VAR
	fbDriveControl 		: FB_DriveControl;
	fResult 			: REAL;
	fExpected 			: REAL;
END_VAR
TEST('Test Property: fAccMax');
fExpected := 10;
fbDriveControl.fAccMax := fExpected;
fResult := fbDriveControl.fAccMax;

AssertEquals(Expected := fExpected,
             Actual := fResult,
             Message := 'Property value is not correct');
TEST_FINISHED();

TEST('Test Property: fPositionLimitMin');
fExpected := 10;
fbDriveControl.fPositionLimitMin := fExpected;
fResult := fbDriveControl.fPositionLimitMin;

AssertEquals(Expected := fExpected,
             Actual := fResult,
             Message := 'Property value is not correct');
TEST_FINISHED();

TEST('Test Property: fPositionLimitMax');
fExpected := 10;
fbDriveControl.fPositionLimitMax := fExpected;
fResult := fbDriveControl.fPositionLimitMax;

AssertEquals(Expected := fExpected,
             Actual := fResult,
             Message := 'Property value is not correct');
TEST_FINISHED();

TEST('Test Property: fTolerance');
fExpected := 10;
fbDriveControl.fTolerance := fExpected;
fResult := fbDriveControl.fTolerance;

AssertEquals(Expected := fExpected,
             Actual := fResult,
             Message := 'Property value is not correct');
TEST_FINISHED();

TEST('Test Property: fPosition');
fExpected := 10;
fbDriveControl.fPosition := fExpected;
fResult := fbDriveControl.fPosition;

AssertEquals(Expected := fExpected,
             Actual := fResult,
             Message := 'Property value is not correct');
TEST_FINISHED();
END_METHOD

METHOD TestStop : REFERENCE TO FB_Test
VAR
	fbDriveControl 		: FB_DriveControl;
	nCycleCount 		: INT;
	bResult 			: BOOL;
	fResult 			: REAL;
	fExpected 			: REAL;
END_VAR
TEST('Stop');

fbDriveControl.fVelocity := -10; 

bResult := fbDriveControl.bIsMoving;
AssertTrue(bResult, 'Expected Drive in motion');

FOR nCycleCount := 0 TO 10 DO
    fbDriveControl.Stop(1E6);
END_FOR

bResult := fbDriveControl.bIsMoving;
AssertFalse(bResult, 'Expected Drive is stopped');

fExpected := 0;
fResult := fbDriveControl.fVelocity;
AssertEquals(Expected := fExpected,
             Actual := fResult,
             Message := 'fVelocity value is not correct');

TEST_FINISHED();
END_METHOD

END_FUNCTION_BLOCK

// Tests/Components/FB_Heater_Test
FUNCTION_BLOCK FB_Heater_Test EXTENDS TcUnit.FB_TestSuite

TestState();
TestLimits();
TestValueChange();

METHOD TestLimits : REFERENCE TO FB_Test
VAR
	fbHeater : FB_Heater(0);
END_VAR
TEST('Limit Min FALSE');
fbHeater.fHeatingSpeed := 0;
fbHeater.fCoolingSpeed := 0;
fbHeater.fLimitMin := 20;
fbHeater.fValue := 30;

fbHeater();

AssertFALSE(fbHeater.bIsLimitMin, 'State is not correct');	 
TEST_FINISHED();

TEST('Limit Min TRUE');
fbHeater.fHeatingSpeed := 0;
fbHeater.fCoolingSpeed := 0;
fbHeater.fLimitMin := 20;
fbHeater.fValue := 20;

fbHeater();

AssertTRUE(fbHeater.bIsLimitMin, 'State is not correct');	 
TEST_FINISHED();

TEST('Limit Max FALSE');
fbHeater.fHeatingSpeed := 0;
fbHeater.fCoolingSpeed := 0;
fbHeater.fLimitMax := 60;
fbHeater.fValue := 59.9999;

fbHeater();

AssertFALSE(fbHeater.bIsLimitMax, 'State is not correct');	 
TEST_FINISHED();

TEST('Limit Max TRUE');
fbHeater.fHeatingSpeed := 0;
fbHeater.fCoolingSpeed := 0;
fbHeater.fLimitMax := 60;
fbHeater.fValue := 60;

fbHeater();

AssertTRUE(fbHeater.bIsLimitMax, 'State is not correct');	 
TEST_FINISHED();
END_METHOD

METHOD TestState : REFERENCE TO FB_Test
VAR
	fbHeater : FB_Heater(0);
END_VAR
TEST('State Enable');
fbHeater.bEnable := TRUE;	
fbHeater();
AssertTRUE(fbHeater.bEnabled, 'State is not correct');	 
TEST_FINISHED();

TEST('State Disable');
fbHeater.bEnable := TRUE;	
fbHeater();
fbHeater.bEnable := FALSE;
fbHeater();	
AssertFALSE(fbHeater.bEnabled, 'State is not correct');	 
TEST_FINISHED();
END_METHOD

METHOD TestValueChange : REFERENCE TO FB_Test
VAR
	fbHeater : FB_Heater(0);
	fResult : REAL;	
	fExpected : REAL;
	bExpected : BOOL;
	fInitValue : REAL;
	nCycleCount : INT;
END_VAR
TEST('Value Up Disable');

fInitValue := 30;

fbHeater.bEnable := FALSE;
fbHeater.fValue := fInitValue;
fbHeater.fHeatingSpeed := 10;
fbHeater.fCoolingSpeed := 0;

fbHeater();

fResult := fbHeater.fValue;
fExpected := fInitValue;

AssertEquals(Expected := fExpected,
             Actual := fResult,
             Message := 'Result value is not correct');	
	 
TEST_FINISHED();


TEST('Value Up Enable');

fInitValue := 30;

fbHeater.bEnable := TRUE;
fbHeater.fValue := fInitValue;
fbHeater.fHeatingSpeed := 10;
fbHeater.fCoolingSpeed := 0;

fbHeater();

fResult := fbHeater.fValue;
fExpected := fInitValue + 10 * GVL_Core.fbSystem.fDeltaTime;

AssertEquals(Expected := fExpected,
             Actual := fResult,
             Message := 'Result value is not correct');	
	 
TEST_FINISHED();


TEST('Value Down Disable');

fInitValue := 30;

fbHeater.bEnable := FALSE;
fbHeater.fValue := fInitValue;
fbHeater.fHeatingSpeed := 10;
fbHeater.fCoolingSpeed := 0;

fbHeater();

fResult := fbHeater.fValue;
fExpected := fInitValue;

AssertEquals(Expected := fExpected,
             Actual := fResult,
             Message := 'Result value is not correct');	
	 
TEST_FINISHED();


TEST('Value Down Enable');

fInitValue := 30;

fbHeater.bEnable := TRUE;
fbHeater.fValue := fInitValue;
fbHeater.fHeatingSpeed := 20;
fbHeater.fCoolingSpeed := 30;

fbHeater();

fResult := fbHeater.fValue;
fExpected := fInitValue - 10 * GVL_Core.fbSystem.fDeltaTime;

AssertEquals(Expected := fExpected,
             Actual := fResult,
             Message := 'Result value is not correct');	
	 
TEST_FINISHED();

TEST('Value Cooling');

fInitValue := 30;

fbHeater.bEnable := FALSE;
fbHeater.fValue := fInitValue;
fbHeater.fHeatingSpeed := 0;
fbHeater.fCoolingSpeed := 10;

fbHeater();

fResult := fbHeater.fValue;
fExpected := fInitValue - 10 * GVL_Core.fbSystem.fDeltaTime;

AssertEquals(Expected := fExpected,
             Actual := fResult,
             Message := 'Result value is not correct');	
	 
TEST_FINISHED();
END_METHOD

END_FUNCTION_BLOCK

// Tests/Components/FB_MoveAbsolute_Test
FUNCTION_BLOCK FB_MoveAbsolute_Test EXTENDS TcUnit.FB_TestSuite

TestCaseMoveTo('Set Init', fInitPosition := 0, fInitVelocity := 0, fPosition := 0, fVelocity := 100, fAcceleration := 1E+6, fDeceleration := 1E+6, TRUE);

TestCaseMoveTo('Set Valid Motion_1', fInitPosition := 0, fInitVelocity := 0, fPosition := 1, fVelocity := 1000, fAcceleration := 1E+6, fDeceleration := 1E+6, TRUE);
TestCaseMoveTo('Set Valid Motion_2', fInitPosition := 0, fInitVelocity := 0, fPosition := 10, fVelocity := 1000, fAcceleration := 1E+6, fDeceleration := 1E+6, TRUE);
TestCaseMoveTo('Set Valid Motion_3', fInitPosition := 0, fInitVelocity := 0, fPosition := 100, fVelocity := 1000, fAcceleration := 1E+6, fDeceleration := 1E+6, FALSE);
TestCaseMoveTo('Set Valid Motion_4', fInitPosition := 0, fInitVelocity := 0, fPosition := 1000, fVelocity := 1000, fAcceleration := 1E+6, fDeceleration := 1E+6, FALSE);

TestCaseMoveTo('Set 2Zone Motion_1', fInitPosition := -5, fInitVelocity := 0, fPosition := 1, fVelocity := 1000, fAcceleration := 1E+6, fDeceleration := 1E+6, TRUE);
TestCaseMoveTo('Set 2Zone Motion_2', fInitPosition := -5, fInitVelocity := 0, fPosition := 5, fVelocity := 1000, fAcceleration := 1E+6, fDeceleration := 1E+6, TRUE);
TestCaseMoveTo('Set 2Zone Motion_3', fInitPosition := 5, fInitVelocity := 0, fPosition := -1, fVelocity := 1000, fAcceleration := 1E+6, fDeceleration := 1E+6, TRUE);
TestCaseMoveTo('Set 2Zone Motion_4', fInitPosition := 5, fInitVelocity := 0, fPosition := -5, fVelocity := 1000, fAcceleration := 1E+6, fDeceleration := 1E+6, TRUE);

TestCaseMoveTo('Set Dirty Motion_1', fInitPosition := 0, fInitVelocity := 0, fPosition := 1, fVelocity := -1000, fAcceleration := -1E+6, fDeceleration := -1E+6, TRUE);
TestCaseMoveTo('Set Dirty Motion_2', fInitPosition := 0, fInitVelocity := 0, fPosition := 10, fVelocity := -1000, fAcceleration := -1E+6, fDeceleration := -1E+6, TRUE);
TestCaseMoveTo('Set Dirty Motion_3', fInitPosition := 0, fInitVelocity := 0, fPosition := 100, fVelocity := -1000, fAcceleration := -1E+6, fDeceleration := -1E+6, FALSE);
TestCaseMoveTo('Set Dirty Motion_4', fInitPosition := 0, fInitVelocity := 0, fPosition := 1000, fVelocity := -1000, fAcceleration := -1E+6, fDeceleration := -1E+6, FALSE);

TestCaseMoveTo('Set Init Velocity_1', fInitPosition := 0, fInitVelocity := 1000, fPosition := 1, fVelocity := 1000, fAcceleration := 1E+6, fDeceleration := 1E+6, TRUE);
TestCaseMoveTo('Set Init Velocity_2', fInitPosition := 0, fInitVelocity := 1000, fPosition := 10, fVelocity := 1000, fAcceleration := 1E+6, fDeceleration := 1E+6, TRUE);
TestCaseMoveTo('Set Init Velocity_3', fInitPosition := 0, fInitVelocity := 1000, fPosition := 100, fVelocity := 1000, fAcceleration := 1E+6, fDeceleration := 1E+6, FALSE);
TestCaseMoveTo('Set Init Velocity_4', fInitPosition := 0, fInitVelocity := 1000, fPosition := 1000, fVelocity := 1000, fAcceleration := 1E+6, fDeceleration := 1E+6, FALSE);

TestCaseMoveTo('Set Init Position_1', fInitPosition := 1, fInitVelocity := 1000, fPosition := 1, fVelocity := 1000, fAcceleration := 1E+6, fDeceleration := 1E+6, TRUE);
TestCaseMoveTo('Set Init Position_2', fInitPosition := 10, fInitVelocity := 1000, fPosition := 10, fVelocity := 1000, fAcceleration := 1E+6, fDeceleration := 1E+6, TRUE);
TestCaseMoveTo('Set Init Position_3', fInitPosition := 100, fInitVelocity := 1000, fPosition := 100, fVelocity := 1000, fAcceleration := 1E+6, fDeceleration := 1E+6, TRUE);
TestCaseMoveTo('Set Init Position_4', fInitPosition := 1000, fInitVelocity := 1000, fPosition := 1000, fVelocity := 1000, fAcceleration := 1E+6, fDeceleration := 1E+6, TRUE);

METHOD TestCaseMoveTo : REFERENCE TO FB_Test
VAR_INPUT
	sName 				: T_MaxString;
	fInitPosition 		: REAL;
	fInitVelocity 		: REAL;
	fPosition 			: REAL;	
	fVelocity 			: REAL; 
	fAcceleration 		: REAL; 
	fDeceleration 		: REAL;	
	bExpected 			: BOOL;
END_VAR

VAR
	fbMoveAbsolute 		: FB_MoveAbsolute;
	nCycleCount 		: INT;
	bResult 			: BOOL;
	fResult 			: REAL;
	fVel 				: REAL;
	fExpectedVel 		: REAL := 0;
END_VAR
TEST(sName);

fbMoveAbsolute.fPosition := fInitPosition;
fbMoveAbsolute.fVelocity := fInitVelocity;

FOR nCycleCount := 0 TO 10 DO
    fbMoveAbsolute( fTargetPosition:= fPosition, 
					fTargetVelocity := fVelocity, 
					fAccMax := fAcceleration, 
					fDecMax := fDeceleration);
END_FOR

bResult := fbMoveAbsolute.bIsReached;
fResult := fbMoveAbsolute.fPosition;
fVel := fbMoveAbsolute.fVelocity;

AssertEquals(Expected := bExpected,
             Actual := bResult,
             Message := 'Value is not reached');

IF bExpected THEN
	AssertEquals(Expected := fPosition,
             Actual := fResult,
             Message := 'Position value is not correct');	
	AssertEquals(Expected := fExpectedVel,
             Actual := fVel,
             Message := 'Velocity value is not correct');	
END_IF
	 
TEST_FINISHED();
END_METHOD

END_FUNCTION_BLOCK

// Tests/Components/FB_MoveVelocity_Test
FUNCTION_BLOCK FB_MoveVelocity_Test EXTENDS TcUnit.FB_TestSuite

TestCaseMove('Set Init',0, 0, 1000, 1000, TRUE);

TestCaseMove('Set Valid Motion_1',0, 1000, 1000, 1000, FALSE);
TestCaseMove('Set Valid Motion_2',0, 100, 1000, 1000, FALSE);
TestCaseMove('Set Valid Motion_3',0, 10, 1000, 1000, TRUE);	
TestCaseMove('Set Valid Motion_4',0, -1000, -1000, -1000, FALSE);
TestCaseMove('Set Valid Motion_5',0, -100, -1000, -1000, FALSE);
TestCaseMove('Set Valid Motion_6',0, -10, -1000, -1000, TRUE);

TestCaseMove('Set 2Zone Motion_1',-5, 1000, 1000, 1000, FALSE);
TestCaseMove('Set 2Zone Motion_2',-5, 100, 1000, 1000, FALSE);
TestCaseMove('Set 2Zone Motion_3',-5, 10, 2000, 2000, TRUE);	
TestCaseMove('Set 2Zone Motion_4',5, -1000, -1000, -1000, FALSE);
TestCaseMove('Set 2Zone Motion_5',5, -100, -1000, -1000, FALSE);
TestCaseMove('Set 2Zone Motion_6',5, -10, -2000, -2000, TRUE);

TestCaseMove('Set Dirty Motion_1',0, 10, 0.001, 0.001, FALSE);
TestCaseMove('Set Dirty Motion_2',0, 10, 0, 0, FALSE);
TestCaseMove('Set Dirty Motion_3',0, 10, 1E+12, 1E+12, TRUE);	
TestCaseMove('Set Dirty Motion_4',0, -1E+3, 1E+12, 1E+12, TRUE);	

TestCaseMove('Set Dirty ACC/DEC_1',0, 1000, -1000, -1000, FALSE);
TestCaseMove('Set Dirty ACC/DEC_2',0, 100, -1000, -1000, FALSE);
TestCaseMove('Set Dirty ACC/DEC_3',0, 10, -1000, -1000, TRUE);
TestCaseMove('Set Dirty ACC/DEC_4',0, -1000, 1000, 1000, FALSE);
TestCaseMove('Set Dirty ACC/DEC_5',0, -100, 1000, 1000, FALSE);
TestCaseMove('Set Dirty ACC/DEC_6',0, -10, 1000, 1000, TRUE);

METHOD TestCaseMove
VAR_INPUT
	sName 				: T_MaxString;
	fInitVelocity 		: REAL;
	fVelocity 			: REAL;
	fAcceleration 		: REAL;
	fDeceleration 		: REAL;
	bExpected 			: BOOL;
END_VAR

VAR
	fbMoveVelocity 		: FB_MoveVelocity;
	nCycleCount 		: INT;
	bResult 			: BOOL;
	fResult 			: REAL;
	fAcc 				: REAL;
	fExpectedAcc 		: REAL := 0;
END_VAR
TEST(sName);
	
fbMoveVelocity.fVelocity := fInitVelocity;

FOR nCycleCount := 0 TO 10 DO
    fbMoveVelocity(fTargetVelocity := fVelocity, fAccMax := fAcceleration, fDecMax := fDeceleration);
END_FOR;

bResult := fbMoveVelocity.bIsReached;
fResult := fbMoveVelocity.fVelocity;
fAcc := fbMoveVelocity.fAcc;

AssertEquals(Expected := bExpected,
             Actual := bResult,
             Message := 'Value is not reached');	
			 
IF bExpected THEN
	AssertEquals(Expected := fVelocity,
             Actual := fResult,
             Message := 'Velocity value is not correct');	
	AssertEquals(Expected := fExpectedAcc,
             Actual := fAcc,
             Message := 'Acc value is not correct');	
END_IF
	 
TEST_FINISHED();
END_METHOD

END_FUNCTION_BLOCK

// Tests/Devices/FB_Button_Test
FUNCTION_BLOCK FB_Button_Test EXTENDS TcUnit.FB_TestSuite
VAR
	fbButton : FB_Button;
	nExpected : BYTE;
	nResult : BYTE;
	bExpected : BOOL;
	bResult : BOOL;
END_VAR

TEST('Set bEnable TRUE');			 
fbButton.bEnable := TRUE; 
fbButton();
nExpected := 1;
nResult := fbButton.GetControl();
AssertEquals(Expected := nExpected,
             Actual := nResult,
             Message := 'Control value is not correct');	 
TEST_FINISHED();

TEST('Set bEnable FALSE');			 
fbButton.bEnable := FALSE; 
fbButton();
nExpected := 0;
nResult := fbButton.GetControl();
AssertEquals(Expected := nExpected,
             Actual := nResult,
             Message := 'Control value is not correct');	 
TEST_FINISHED();


TEST('Get bValue FALSE');
fbButton.SetStatus(0);
fbButton();
bExpected := FALSE;
bResult := fbButton.bValue;

AssertEquals(Expected := bExpected,
             Actual := bResult,
             Message := 'Value is not correct');	
TEST_FINISHED();

TEST('Get bValue TRUE');	
fbButton.SetStatus(1);
fbButton();
bExpected := 1;
bResult := fbButton.bValue;
AssertEquals(Expected := bExpected,
             Actual := bResult,
             Message := 'Control value is not correct');	 
TEST_FINISHED();

END_FUNCTION_BLOCK

// Tests/Devices/FB_Cylinder_Test
FUNCTION_BLOCK FB_Cylinder_Test EXTENDS TcUnit.FB_TestSuite
VAR
	fbCylinder : FB_Cylinder;
	nExpected : BYTE;
	nResult : BYTE;
	bExpected : BOOL;
	bResult : BOOL;
END_VAR

TEST('bRetract FALSE');
fbCylinder.bRetract := FALSE;
fbCylinder();
bExpected := FALSE;
nResult := fbCylinder.GetControl();
bResult := nResult.0;

AssertEquals(Expected := bExpected,
             Actual := bResult,
             Message := 'Control value is not correct');	
TEST_FINISHED();

TEST('bRetract TRUE');
fbCylinder.bRetract := TRUE;
fbCylinder();
bExpected := TRUE;
nResult := fbCylinder.GetControl();
bResult := nResult.0;

AssertEquals(Expected := bExpected,
             Actual := bResult,
             Message := 'Control value is not correct');	
TEST_FINISHED();

TEST('bExtend FALSE');
fbCylinder.bExtend := FALSE;
fbCylinder();
bExpected := FALSE;
nResult := fbCylinder.GetControl();
bResult := nResult.1;

AssertEquals(Expected := bExpected,
             Actual := bResult,
             Message := 'Control value is not correct');	
TEST_FINISHED();

TEST('bExtend TRUE');
fbCylinder.bExtend := TRUE;
fbCylinder();
bExpected := TRUE;
nResult := fbCylinder.GetControl();
bResult := nResult.1;

AssertEquals(Expected := bExpected,
             Actual := bResult,
             Message := 'Control value is not correct');	
TEST_FINISHED();

TEST('bRetracted FALSE');
fbCylinder.SetStatus(0);
fbCylinder();
bExpected := FALSE;
bResult := fbCylinder.bRetracted;

AssertEquals(Expected := bExpected,
             Actual := bResult,
             Message := 'Control value is not correct');	
TEST_FINISHED();

TEST('bRetracted TRUE');
fbCylinder.SetStatus(1);
fbCylinder();
bExpected := TRUE;
bResult := fbCylinder.bRetracted;

AssertEquals(Expected := bExpected,
             Actual := bResult,
             Message := 'Control value is not correct');	
TEST_FINISHED();

TEST('bExtended FALSE');
fbCylinder.SetStatus(0);
fbCylinder();
bExpected := FALSE;
bResult := fbCylinder.bExtended;

AssertEquals(Expected := bExpected,
             Actual := bResult,
             Message := 'Control value is not correct');	
TEST_FINISHED();

TEST('bExtended TRUE');
fbCylinder.SetStatus(2);
fbCylinder();
bExpected := TRUE;
bResult := fbCylinder.bExtended;

AssertEquals(Expected := bExpected,
             Actual := bResult,
             Message := 'Control value is not correct');	
TEST_FINISHED();

END_FUNCTION_BLOCK

// Tests/Devices/FB_Device_Test
FUNCTION_BLOCK FB_Device_Test EXTENDS TcUnit.FB_TestSuite
VAR
	fbDevice : FB_Device;
	nExpected : BYTE;
	nResult : BYTE;
END_VAR

TEST('Set nControl');
nExpected := 255;
fbDevice.nControl := nExpected;
fbDevice();
nResult := fbDevice.GetControl();

AssertEquals(Expected := nExpected,
             Actual := nResult,
             Message := 'Value is not correct');	
TEST_FINISHED();

TEST('Get nStatus');
nExpected := 255;
fbDevice.SetStatus(nExpected);
fbDevice();
nResult := fbDevice.nStatus;

AssertEquals(Expected := nExpected,
             Actual := nResult,
             Message := 'Value is not correct');	
TEST_FINISHED();

END_FUNCTION_BLOCK

// Tests/Devices/FB_DeviceByte_Test
FUNCTION_BLOCK FB_DeviceByte_Test EXTENDS TcUnit.FB_TestSuite
VAR
	fbDevice : FB_DeviceByte;
	nExpected : BYTE;
	nResult : BYTE;
END_VAR

TEST('Set nControl');
nExpected := 255;
fbDevice.nControl := nExpected;
fbDevice();
nResult := fbDevice.GetControl();

AssertEquals(Expected := nExpected,
             Actual := nResult,
             Message := 'Value is not correct');	
TEST_FINISHED();

TEST('Set nDataIn');
nExpected := 255;
fbDevice.nControlData := nExpected;
fbDevice();
nResult := fbDevice.GetLinkControlData();

AssertEquals(Expected := nExpected,
             Actual := nResult,
             Message := 'Value is not correct');	
TEST_FINISHED();

TEST('Get nStatus');
nExpected := 255;
fbDevice.SetStatus(nExpected);
fbDevice();
nResult := fbDevice.nStatus;

AssertEquals(Expected := nExpected,
             Actual := nResult,
             Message := 'Value is not correct');	
TEST_FINISHED();

TEST('Get nDataOut');
nExpected := 255;
fbDevice.SetLinkStatusData(nExpected);
fbDevice();
nResult := fbDevice.nStatusData;

AssertEquals(Expected := nExpected,
             Actual := nResult,
             Message := 'Value is not correct');	
TEST_FINISHED();

END_FUNCTION_BLOCK

// Tests/Devices/FB_DeviceDWord_Test
FUNCTION_BLOCK FB_DeviceDWord_Test EXTENDS TcUnit.FB_TestSuite
VAR
	fbDevice : FB_DeviceDWord;
	nExpected : DWORD;
	nResult : DWORD;
	nValue : DWORD := 16#FFAA;
END_VAR

TEST('Set nControl');
nExpected := 255;
fbDevice.nControl := 255;
fbDevice();
nResult := fbDevice.GetControl();

AssertEquals(Expected := nExpected,
             Actual := nResult,
             Message := 'Value is not correct');	
TEST_FINISHED();

TEST('Set nDataIn');
nExpected := nValue;
fbDevice.nControlData := nExpected;
fbDevice();
nResult := fbDevice.GetLinkControlData();

AssertEquals(Expected := nExpected,
             Actual := nResult,
             Message := 'Value is not correct');	
TEST_FINISHED();

TEST('Get nStatus');
nExpected := 255;
fbDevice.SetStatus(255);
fbDevice();
nResult := fbDevice.nStatus;

AssertEquals(Expected := nExpected,
             Actual := nResult,
             Message := 'Value is not correct');	
TEST_FINISHED();

TEST('Get nDataOut');
nExpected := nValue;
fbDevice.SetLinkStatusData(nExpected);
fbDevice();
nResult := fbDevice.nStatusData;

AssertEquals(Expected := nExpected,
             Actual := nResult,
             Message := 'Value is not correct');	
TEST_FINISHED();

END_FUNCTION_BLOCK

// Tests/Devices/FB_DeviceLWord_Test
FUNCTION_BLOCK FB_DeviceLWord_Test EXTENDS TcUnit.FB_TestSuite
VAR
	fbDevice : FB_DeviceLWord;
	nExpected : LWORD;
	nResult : LWORD;
	nValue : LWORD := 16#FFAABBCC;
END_VAR

TEST('Set nControl');
nExpected := 255;
fbDevice.nControl := 255;
fbDevice();
nResult := fbDevice.GetControl();

AssertEquals(Expected := nExpected,
             Actual := nResult,
             Message := 'Value is not correct');	
TEST_FINISHED();

TEST('Set nDataIn');
nExpected := nValue;
fbDevice.nControlData := nExpected;
fbDevice();
nResult := fbDevice.GetLinkControlData();

AssertEquals(Expected := nExpected,
             Actual := nResult,
             Message := 'Value is not correct');	
TEST_FINISHED();

TEST('Get nStatus');
nExpected := 255;
fbDevice.SetStatus(255);
fbDevice();
nResult := fbDevice.nStatus;

AssertEquals(Expected := nExpected,
             Actual := nResult,
             Message := 'Value is not correct');	
TEST_FINISHED();

TEST('Get nDataOut');
nExpected := nValue;
fbDevice.SetLinkStatusData(nExpected);
fbDevice();
nResult := fbDevice.nStatusData;

AssertEquals(Expected := nExpected,
             Actual := nResult,
             Message := 'Value is not correct');	
TEST_FINISHED();

END_FUNCTION_BLOCK

// Tests/Devices/FB_DeviceReal_Test
FUNCTION_BLOCK FB_DeviceReal_Test EXTENDS TcUnit.FB_TestSuite
VAR
	fbDevice : FB_DeviceReal;
	fExpected : REAL;
	fResult : REAL;
	fValue : REAL := 16#FF;
END_VAR

TEST('Set nControl');
fExpected := 255;
fbDevice.nControl := 255;
fbDevice();
fResult := fbDevice.GetControl();

AssertEquals(Expected := fExpected,
             Actual := fResult,
             Message := 'Value is not correct');	
TEST_FINISHED();

TEST('Set nDataIn_1');
fExpected := 1000;
fbDevice.fControlData := fExpected;
fbDevice();
fResult := fbDevice.GetLinkControlData();

AssertEquals(Expected := fExpected,
             Actual := fResult,
             Message := 'Value is not correct');	
TEST_FINISHED();

TEST('Set nDataIn_2');
fExpected := -1000;
fbDevice.fControlData := fExpected;
fbDevice();
fResult := fbDevice.GetLinkControlData();

AssertEquals(Expected := fExpected,
             Actual := fResult,
             Message := 'Value is not correct');	
TEST_FINISHED();

TEST('Get nStatus');
fExpected := 255;
fbDevice.SetStatus(255);
fbDevice();
fResult := fbDevice.nStatus;

AssertEquals(Expected := fExpected,
             Actual := fResult,
             Message := 'Value is not correct');	
TEST_FINISHED();

TEST('Get nDataOut_1');
fExpected := 1000;
fbDevice.SetLinkStatusData(fExpected);
fbDevice();
fResult := fbDevice.fStatusData;

AssertEquals(Expected := fExpected,
             Actual := fResult,
             Message := 'Value is not correct');	
TEST_FINISHED();

TEST('Get nDataOut_2');
fExpected := -1000;
fbDevice.SetLinkStatusData(fExpected);
fbDevice();
fResult := fbDevice.fStatusData;

AssertEquals(Expected := fExpected,
             Actual := fResult,
             Message := 'Value is not correct');	
TEST_FINISHED();

END_FUNCTION_BLOCK

// Tests/Devices/FB_DeviceWord_Test
FUNCTION_BLOCK FB_DeviceWord_Test EXTENDS TcUnit.FB_TestSuite
VAR
	fbDevice : FB_DeviceWord;
	nExpected : WORD;
	nResult : WORD;
	nValue : WORD := 16#FF;
END_VAR

TEST('Set nControl');
nExpected := 255;
fbDevice.nControl := 255;
fbDevice();
nResult := fbDevice.GetControl();

AssertEquals(Expected := nExpected,
             Actual := nResult,
             Message := 'Value is not correct');	
TEST_FINISHED();

TEST('Set nDataIn');
nExpected := nValue;
fbDevice.nControlData := nExpected;
fbDevice();
nResult := fbDevice.GetLinkControlData();

AssertEquals(Expected := nExpected,
             Actual := nResult,
             Message := 'Value is not correct');	
TEST_FINISHED();

TEST('Get nStatus');
nExpected := 255;
fbDevice.SetStatus(255);
fbDevice();
nResult := fbDevice.nStatus;

AssertEquals(Expected := nExpected,
             Actual := nResult,
             Message := 'Value is not correct');	
TEST_FINISHED();

TEST('Get nDataOut');
nExpected := nValue;
fbDevice.SetLinkStatusData(nExpected);
fbDevice();
nResult := fbDevice.nStatusData;

AssertEquals(Expected := nExpected,
             Actual := nResult,
             Message := 'Value is not correct');	
TEST_FINISHED();

END_FUNCTION_BLOCK

// Tests/Devices/FB_Drive_Test
FUNCTION_BLOCK FB_Drive_Test EXTENDS TcUnit.FB_TestSuite
VAR
	fbDrive : FB_Drive;
	nExpectedByte : BYTE;
	nResultByte : BYTE;
	fExpectedReal : REAL;
	fResultReal : REAL;
END_VAR

TEST('Set nControl');
nExpectedByte := 255;
fbDrive.nControl := nExpectedByte;
fbDrive();
nResultByte := fbDrive.GetControl();

AssertEquals(Expected := nExpectedByte,
             Actual := nResultByte,
             Message := 'Value is not correct');	
TEST_FINISHED();

TEST('Get nStatus');
nExpectedByte := 255;
fbDrive.SetStatus(nExpectedByte);
fbDrive();
nResultByte := fbDrive.nStatus;

AssertEquals(Expected := nExpectedByte,
             Actual := nResultByte,
             Message := 'Value is not correct');	
TEST_FINISHED();

TEST('Set fTargetValue_1');
fExpectedReal := 1000;
fbDrive.fTargetValue := fExpectedReal;
fbDrive();
fResultReal := fbDrive.GetLinkControlData();

AssertEquals(Expected := fExpectedReal,
             Actual := fResultReal,
             Message := 'Value is not correct');	
TEST_FINISHED();

TEST('Set fTargetValue_2');
fExpectedReal := -1000;
fbDrive.fTargetValue := fExpectedReal;
fbDrive();
fResultReal := fbDrive.GetLinkControlData();

AssertEquals(Expected := fExpectedReal,
             Actual := fResultReal,
             Message := 'Value is not correct');	
TEST_FINISHED();

TEST('Get fActualValue_1');
fExpectedReal := 1000;
fbDrive.SetLinkStatusData(fExpectedReal);
fbDrive();
fResultReal := fbDrive.fActualValue;

AssertEquals(Expected := fExpectedReal,
             Actual := fResultReal,
             Message := 'Value is not correct');	
TEST_FINISHED();

TEST('Get fActualValue_2');
fExpectedReal := -1000;
fbDrive.SetLinkStatusData(fExpectedReal);
fbDrive();
fResultReal := fbDrive.fActualValue;

AssertEquals(Expected := fExpectedReal,
             Actual := fResultReal,
             Message := 'Value is not correct');	
TEST_FINISHED();

END_FUNCTION_BLOCK

// Tests/Devices/FB_Lamp_Test
FUNCTION_BLOCK FB_Lamp_Test EXTENDS TcUnit.FB_TestSuite
VAR
	fbLamp : FB_Lamp;
	nExpected : BYTE;
	nResult : BYTE;
	bExpected : BOOL;
	bResult : BOOL;
END_VAR

TEST('Set bEnable TRUE');			 
fbLamp.bEnable := TRUE; 
fbLamp();
nExpected := 1;
nResult := fbLamp.GetControl();
AssertEquals(Expected := nExpected,
             Actual := nResult,
             Message := 'Control value is not correct');	 
TEST_FINISHED();

TEST('Set bEnable FALSE');			 
fbLamp.bEnable := FALSE; 
fbLamp();
nExpected := 0;
nResult := fbLamp.GetControl();
AssertEquals(Expected := nExpected,
             Actual := nResult,
             Message := 'Control value is not correct');	 
TEST_FINISHED();

END_FUNCTION_BLOCK

// Tests/Devices/FB_Lock_Test
FUNCTION_BLOCK FB_Lock_Test EXTENDS TcUnit.FB_TestSuite
VAR
	fbLock : FB_Lock;
	nExpected : BYTE;
	nResult : BYTE;
	bExpected : BOOL;
	bResult : BOOL;
END_VAR

TEST('Set bEnable TRUE');			 
fbLock.bLock := TRUE; 
fbLock();
nExpected := 1;
nResult := fbLock.GetControl();
AssertEquals(Expected := nExpected,
             Actual := nResult,
             Message := 'Control value is not correct');	 
TEST_FINISHED();

TEST('Set bEnable FALSE');			 
fbLock.bLock := FALSE; 
fbLock();
nExpected := 0;
nResult := fbLock.GetControl();
AssertEquals(Expected := nExpected,
             Actual := nResult,
             Message := 'Value is not correct');	 
TEST_FINISHED();


TEST('Get bClosed FALSE');
fbLock.SetStatus(0);
fbLock();
bExpected := FALSE;
bResult := fbLock.bClosed;

AssertEquals(Expected := bExpected,
             Actual := bResult,
             Message := 'Value is not correct');	
TEST_FINISHED();

TEST('Get bClosed TRUE');	
fbLock.SetStatus(1);
fbLock();
bExpected := 1;
bResult := fbLock.bClosed;
AssertEquals(Expected := bExpected,
             Actual := bResult,
             Message := 'Value is not correct');	 
TEST_FINISHED();

TEST('Get bLocked FALSE');
fbLock.SetStatus(0);
fbLock();
bExpected := FALSE;
bResult := fbLock.bLocked;

AssertEquals(Expected := bExpected,
             Actual := bResult,
             Message := 'Value is not correct');	
TEST_FINISHED();

TEST('Get bLocked TRUE');	
fbLock.SetStatus(2);
fbLock();
bExpected := 1;
bResult := fbLock.bLocked;
AssertEquals(Expected := bExpected,
             Actual := bResult,
             Message := 'Value is not correct');	 
TEST_FINISHED();

TEST('Set nDataIn');
nExpected := 255;
fbLock.nControlData := nExpected;
fbLock();
nResult := fbLock.GetLinkControlData();

AssertEquals(Expected := nExpected,
             Actual := nResult,
             Message := 'Value is not correct');	
TEST_FINISHED();

TEST('Get nDataOut');
nExpected := 255;
fbLock.SetLinkStatusData(nExpected);
fbLock();
nResult := fbLock.nStatusData;

AssertEquals(Expected := nExpected,
             Actual := nResult,
             Message := 'Value is not correct');	
TEST_FINISHED();

END_FUNCTION_BLOCK

// Tests/Devices/FB_Panel_Test
FUNCTION_BLOCK FB_Panel_Test EXTENDS TcUnit.FB_TestSuite
VAR
	fbPanel : FB_Panel;
	nExpected : DWORD;
	nResult : DWORD;
	bExpected : BOOL;
	bResult : BOOL;
END_VAR

TEST('Set nDataIn');
nExpected := 255;
fbPanel.nControlData := nExpected;
fbPanel();
nResult := fbPanel.GetLinkControlData();

AssertEquals(Expected := nExpected,
             Actual := nResult,
             Message := 'Value is not correct');	
TEST_FINISHED();

TEST('Get nDataOut');
nExpected := 255;
fbPanel.SetLinkStatusData(nExpected);
fbPanel();
nResult := fbPanel.nStatusData;

AssertEquals(Expected := nExpected,
             Actual := nResult,
             Message := 'Value is not correct');	
TEST_FINISHED();

END_FUNCTION_BLOCK

// Tests/Devices/FB_Reader_Test
FUNCTION_BLOCK FB_Reader_Test EXTENDS TcUnit.FB_TestSuite
VAR
	fbDevice : FB_Reader;
	nExpected : LWORD;
	nResult : LWORD;
	nValue : LWORD := 16#FFAABBCC;
END_VAR

TEST('Set nControl');
nExpected := 255;
fbDevice.nControl := 255;
fbDevice();
nResult := fbDevice.GetControl();

AssertEquals(Expected := nExpected,
             Actual := nResult,
             Message := 'Value is not correct');	
TEST_FINISHED();

TEST('Set nCommand');
nExpected := nValue;
fbDevice.nCommand := nExpected;
fbDevice();
nResult := fbDevice.GetLinkControlData();

AssertEquals(Expected := nExpected,
             Actual := nResult,
             Message := 'Value is not correct');	
TEST_FINISHED();

TEST('Get nStatus');
nExpected := 255;
fbDevice.SetStatus(255);
fbDevice();
nResult := fbDevice.nStatus;

AssertEquals(Expected := nExpected,
             Actual := nResult,
             Message := 'Value is not correct');	
TEST_FINISHED();

TEST('Get nResult');
nExpected := nValue;
fbDevice.SetLinkStatusData(nExpected);
fbDevice();
nResult := fbDevice.nResult;

AssertEquals(Expected := nExpected,
             Actual := nResult,
             Message := 'Value is not correct');	
TEST_FINISHED();

END_FUNCTION_BLOCK

// Tests/Devices/FB_Robot_Test
FUNCTION_BLOCK FB_Robot_Test EXTENDS TcUnit.FB_TestSuite
VAR
	fbRobot : FB_Robot;
	nExpectedByte : BYTE;
	nResultByte : BYTE;
	aExpectedJoints : ARRAY[0..11] OF REAL := [11, 22, 33, 44, 55, 66, 77, 88, 99, 1010, 1111, 1212];	
	aResultJoints : ARRAY[0..11] OF REAL;	
	nJointCount : INT := 12;
END_VAR

TEST('Set nControl');
nExpectedByte := 255;
fbRobot.nControl := nExpectedByte;
fbRobot();
nResultByte := fbRobot.GetControl();

AssertEquals(Expected := nExpectedByte,
             Actual := nResultByte,
             Message := 'Value is not correct');	
TEST_FINISHED();

TEST('Get nStatus');
nExpectedByte := 255;
fbRobot.SetStatus(nExpectedByte);
fbRobot();
nResultByte := fbRobot.nStatus;

AssertEquals(Expected := nExpectedByte,
             Actual := nResultByte,
             Message := 'Value is not correct');	
TEST_FINISHED();

TestSetJoint('Set Joint 1', 0, 100);
TestSetJoint('Set Joint 2', 1, 100);
TestSetJoint('Set Joint 3', 2, 100);
TestSetJoint('Set Joint 4', 3, 100);
TestSetJoint('Set Joint 5', 4, 100);
TestSetJoint('Set Joint 6', 5, 100);
TestSetJoint('Set Joint EXT1', 6, 100);
TestSetJoint('Set Joint EXT2', 7, 100);
TestSetJoint('Set Joint EXT3', 8, 100);
TestSetJoint('Set Joint EXT4', 9, 100);
TestSetJoint('Set Joint EXT5', 10, 100);
TestSetJoint('Set Joint EXT6', 11, 100);

TestGetJoint('Get Joint 1', 0, 100);
TestGetJoint('Get Joint 2', 1, 100);
TestGetJoint('Get Joint 3', 2, 100);
TestGetJoint('Get Joint 4', 3, 100);
TestGetJoint('Get Joint 5', 4, 100);
TestGetJoint('Get Joint 6', 5, 100);
TestGetJoint('Get Joint EXT1', 6, 100);
TestGetJoint('Get Joint EXT2', 7, 100);
TestGetJoint('Get Joint EXT3', 8, 100);
TestGetJoint('Get Joint EXT4', 9, 100);
TestGetJoint('Get Joint EXT5', 10, 100);
TestGetJoint('Get Joint EXT6', 11, 100);

TEST('Set Joints wia Pointer');
fbRobot.ConnectJoints(aExpectedJoints, 12);
fbRobot();
aResultJoints := fbRobot.GetJointsTarget();
AssertEquals(Expected := aExpectedJoints,
             Actual := aResultJoints,
             Message := 'Value is not correct');	
TEST_FINISHED();

METHOD TestGetJoint : BOOL
VAR_INPUT
	sName : T_MaxString;
	nJointIndex : INT;
	fValue : REAL;
END_VAR

VAR
	fbRobot : FB_Robot;	
	fResult : REAL;		
	aExpectedJoints : ARRAY[0..11] OF REAL;
END_VAR
TEST(sName);

aExpectedJoints[nJointIndex] := fValue;
fbRobot.SetJointsStatus(aExpectedJoints);
fbRobot();
fResult := fbRobot.aJointStatus[nJointIndex];

AssertEquals(Expected := fValue,
             Actual := fResult,
             Message := 'Result value is not correct');	
	 
TEST_FINISHED();
END_METHOD

METHOD TestSetJoint : BOOL
VAR_INPUT
	sName : T_MaxString;
	nJointIndex : INT;
	fValue : REAL;
END_VAR

VAR
	fbRobot : FB_Robot;	
	fResult : REAL;		
	aResultJoints : ARRAY[0..11] OF REAL;
END_VAR
TEST(sName);

fbRobot.aJointTarget[nJointIndex] := fValue;
fbRobot();
aResultJoints := fbRobot.GetJointsTarget();
fResult := aResultJoints[nJointIndex];

AssertEquals(Expected := fValue,
             Actual := fResult,
             Message := 'Result value is not correct');	
	 
TEST_FINISHED();
END_METHOD

END_FUNCTION_BLOCK

// Tests/Devices/FB_SensorAnalog_Test
FUNCTION_BLOCK FB_SensorAnalog_Test EXTENDS TcUnit.FB_TestSuite
VAR
	fbSensorAnalog : FB_SensorAnalog;
	nExpectedByte : BYTE;
	nResultByte : BYTE;
	nExpectedUInt : UINT;
	nResultUInt : UINT;
	fExpectedReal : REAL;
	fResultReal : REAL;
END_VAR

TEST('Set nControl');
nExpectedByte := 255;
fbSensorAnalog.nControl := nExpectedByte;
fbSensorAnalog();
nResultByte := fbSensorAnalog.GetControl();

AssertEquals(Expected := nExpectedByte,
             Actual := nResultByte,
             Message := 'Value is not correct');	
TEST_FINISHED();

TEST('Get nStatus');
nExpectedByte := 255;
fbSensorAnalog.SetStatus(nExpectedByte);
fbSensorAnalog();
nResultByte := fbSensorAnalog.nStatus;

AssertEquals(Expected := nExpectedByte,
             Actual := nResultByte,
             Message := 'Value is not correct');	
TEST_FINISHED();


TEST('Get fValue');
fExpectedReal := 50;
nExpectedUInt := 16#8000;
fbSensorAnalog.SetLinkStatusData(fExpectedReal);
fbSensorAnalog();
fResultReal := fbSensorAnalog.fValue;
nResultUInt := fbSensorAnalog.nValue;

AssertEquals(Expected := fExpectedReal,
             Actual := fResultReal,
             Message := 'fValue is not correct');	
AssertEquals(Expected := nExpectedUInt,
             Actual := nResultUInt,
             Message := 'nValue is not correct');
TEST_FINISHED();

END_FUNCTION_BLOCK

// Tests/Devices/FB_SensorBinary_Test
FUNCTION_BLOCK FB_SensorBinary_Test EXTENDS TcUnit.FB_TestSuite
VAR
	fbSensorBinary : FB_SensorBinary;
	nExpected : BYTE;
	nResult : BYTE;
	bExpected : BOOL;
	bResult : BOOL;
END_VAR

TEST('Get bValue FALSE');
fbSensorBinary.SetStatus(0);
fbSensorBinary();
bExpected := FALSE;
bResult := fbSensorBinary.bValue;

AssertEquals(Expected := bExpected,
             Actual := bResult,
             Message := 'Value is not correct');	
TEST_FINISHED();

TEST('Get bValue TRUE');	
fbSensorBinary.SetStatus(1);
fbSensorBinary();
bExpected := 1;
bResult := fbSensorBinary.bValue;
AssertEquals(Expected := bExpected,
             Actual := bResult,
             Message := 'Control value is not correct');	 
TEST_FINISHED();

END_FUNCTION_BLOCK

// Tests/Devices/FB_Switch_Test
FUNCTION_BLOCK FB_Switch_Test EXTENDS TcUnit.FB_TestSuite
VAR
	fbDevice : FB_Switch;
	nExpected : BYTE;
	nResult : BYTE;
END_VAR

TEST('Set nControl');
nExpected := 255;
fbDevice.nControl := nExpected;
fbDevice();
nResult := fbDevice.GetControl();

AssertEquals(Expected := nExpected,
             Actual := nResult,
             Message := 'Value is not correct');	
TEST_FINISHED();

TEST('Get nStatus');
nExpected := 255;
fbDevice.SetStatus(nExpected);
fbDevice();
nResult := fbDevice.nStatus;

AssertEquals(Expected := nExpected,
             Actual := nResult,
             Message := 'Value is not correct');	
TEST_FINISHED();

END_FUNCTION_BLOCK

// Tests/Drives/FB_DS402_Test
FUNCTION_BLOCK FB_DS402_Test EXTENDS TcUnit.FB_TestSuite

TestEnable();
TestEnableSTO();

TestSpeedMode('Speed Mode Target_1', 0, 2000, 0);
TestSpeedMode('Speed Mode Target_2', 40000, 2000, 1000);
TestSpeedMode('Speed Mode Target_3', 80000, 2000, 2000);
TestSpeedMode('Speed Mode Target_4', 100000, 2000, 2000);
TestSpeedMode('Speed Mode Target_5', -40000, 2000, -1000);
TestSpeedMode('Speed Mode Target_6', -80000, 2000, -2000);
TestSpeedMode('Speed Mode Target_7', -100000, 2000, -2000);

TestSpeedDriveFactor('Speed Mode Drive Factor_1', 0, 1, 0);
TestSpeedDriveFactor('Speed Mode Drive Factor_2', 40000, 2, 2000);
TestSpeedDriveFactor('Speed Mode Drive Factor_3', 40000, -2, -2000);
TestSpeedDriveFactor('Speed Mode Drive Factor_4', -40000, 2, -2000);
TestSpeedDriveFactor('Speed Mode Drive Factor_5', -40000, -2, 2000);

TestSpeedModeEncoder('Speed Mode Encoder Value_1', 40000, -0.0001, 1, 10000);
TestSpeedModeEncoder('Speed Mode Encoder Value_2', 40000, -0.001, 1, 1000);
TestSpeedModeEncoder('Speed Mode Encoder Value_3', 40000, 0.001, -10, 10000);
TestSpeedModeEncoder('Speed Mode Encoder Value_4', -40000, -0.0001, -1, -10000);
TestSpeedModeEncoder('Speed Mode Encoder Value_5', -40000, 0.001, -1, -1000);
TestSpeedModeEncoder('Speed Mode Encoder Value_6', -40000, -0.001, 10, -10000);

TestSpeedModeModulo('Speed Mode Modulo Value_1', 40000, 0, 10);
TestSpeedModeModulo('Speed Mode Modulo Value_2', 40000, 3, 1);
TestSpeedModeModulo('Speed Mode Modulo Value_3', 40000, 9, 1);

TestSpeedModeOffset('Speed Mode Position Offset Value_1', 40000, 0, 1);
TestSpeedModeOffset('Speed Mode Position Offset Value_2', 40000, 10, 11);
TestSpeedModeOffset('Speed Mode Position Offset Value_3', 40000, 100, 101);
TestSpeedModeOffset('Speed Mode Position Offset Value_4', 40000, -10, -9);
TestSpeedModeOffset('Speed Mode Position Offset Value_5', 40000, -100, -99);

TestSpeedModeLinkOutput('Link Speed Output Factor_1', 40000, E_ControlMode.Speed, 1, 1000);
TestSpeedModeLinkOutput('Link Speed Output Factor_2', 40000, E_ControlMode.Speed, -1, -1000);
TestSpeedModeLinkOutput('Link Speed Output Factor_3', 40000, E_ControlMode.Speed, 2, 2000);
TestSpeedModeLinkOutput('Link Speed Output Factor_4', 40000, E_ControlMode.Speed, -2, -2000);

TestSpeedModeLinkOutput('Link Position Output Factor_1', 40000, E_ControlMode.Position, 1, 1);
TestSpeedModeLinkOutput('Link Position Output Factor_2', 40000, E_ControlMode.Position, -1, -1);
TestSpeedModeLinkOutput('Link Position Output Factor_3', 40000, E_ControlMode.Position, 2, 2);
TestSpeedModeLinkOutput('Link Position Output Factor_4', 40000, E_ControlMode.Position, -2, -2);

TestPositionMode('Set Target Position_1', 0);
TestPositionMode('Set Target Position_2', 1000);
TestPositionMode('Set Target Position_3', 2000);
TestPositionMode('Set Target Position_4', -1000);
TestPositionMode('Set Target Position_5', -2000);

METHOD EnableSequence : REFERENCE TO FB_Test
VAR_INPUT
	fbDS402 : REFERENCE TO FB_DS402;
END_VAR
fbDS402.stControlData.b0_SwitchOn := FALSE;
fbDS402.stControlData.b1_EnableVoltage := FALSE;
fbDS402.stControlData.b2_QuickStop := FALSE;
fbDS402.stControlData.b3_EnableOperation := FALSE;
fbDS402();

fbDS402.stControlData.b1_EnableVoltage := TRUE;
fbDS402.stControlData.b2_QuickStop := TRUE;
fbDS402();
fbDS402.stControlData.b0_SwitchOn := TRUE;
fbDS402();
fbDS402.stControlData.b3_EnableOperation := TRUE;
fbDS402();
END_METHOD

METHOD TestEnable : BOOL
VAR
	fbDS402 			: FB_DS402;
	nMask 				: WORD;
	nResult 			: WORD;
	bResult 			: BOOL;
	nActualState		: INT;
	nExpectedState		: INT;
END_VAR
TEST('Enable STO FALSE');
fbDS402.bSTO := FALSE;

EnableSequence(fbDS402);

nExpectedState := E_DS402State.S0_NotReadyToSwitchOn;
nActualState := fbDS402.eState;

AssertEquals(Expected := nExpectedState,
             Actual := nActualState,
             Message := 'State is not correct');	 
TEST_FINISHED();
END_METHOD

METHOD TestEnableSTO : BOOL
VAR
	fbDS402 			: FB_DS402;
	nMask 				: WORD;
	nResult 			: WORD;
	bResult 			: BOOL;
	nActualState		: INT;
	nExpectedState		: INT;
END_VAR
TEST('Enable STO TRUE');
fbDS402.bSTO := TRUE;
EnableSequence(fbDS402);

nExpectedState := E_DS402State.S4_OperationEnabled;
nActualState := fbDS402.eState;

AssertEquals(Expected := nExpectedState,
             Actual := nActualState,
             Message := 'State is not correct');	 
TEST_FINISHED();
END_METHOD

METHOD TestPositionMode : BOOL
VAR_INPUT
	sName 				: T_MaxString;
	fTarget				: REAL;	
END_VAR

VAR
	fbDS402 			: FB_DS402;	
	fResult 			: REAL;
END_VAR
TEST(sName);
fbDS402.bSTO := TRUE;
EnableSequence(fbDS402);

fbDS402.stConfig.eControlMode := E_ControlMode.Position;
fbDS402.nTargetValue := REAL_TO_DINT(fTarget * fbDS402.stConfig.fEncoderDenominator / fbDS402.stConfig.fEncoderNumerator);

fbDS402();
fResult := fbDS402.fPosition;

AssertEquals(Expected := fTarget,
             Actual := fResult,
             Message := 'Value is not correct');	 
TEST_FINISHED();
END_METHOD

METHOD TestSpeedDriveFactor : BOOL
VAR_INPUT
	sName 				: T_MaxString;
	nTarget				: DINT;
	fDriveFactor		: REAL;
	fExpected 			: REAL;
END_VAR

VAR
	fbDS402 			: FB_DS402;	
	fResult 			: REAL;
END_VAR
TEST(sName);
fbDS402.bSTO := TRUE;
EnableSequence(fbDS402);

fbDS402.stConfig.eControlMode := E_ControlMode.Speed;
fbDS402.stConfig.fGearFactor := fDriveFactor;
fbDS402.stConfig.fReferenceVelocity := 2000;

fbDS402.nTargetValue := nTarget;

fbDS402();
fResult := fbDS402.fVelocity;

AssertEquals(Expected := fExpected,
             Actual := fResult,
             Message := 'Value is not correct');	 
TEST_FINISHED();
END_METHOD

METHOD TestSpeedMode : BOOL
VAR_INPUT
	sName 				: T_MaxString;
	nTarget				: DINT;
	fReferenceVelocity	: REAL;
	fExpected 			: REAL;
END_VAR

VAR
	fbDS402 			: FB_DS402;	
	fResult 			: REAL;
END_VAR
TEST(sName);
fbDS402.bSTO := TRUE;
EnableSequence(fbDS402);

fbDS402.stConfig.eControlMode := E_ControlMode.Speed;
fbDS402.stConfig.fReferenceVelocity := fReferenceVelocity;

fbDS402.nTargetValue := nTarget;

fbDS402();
fResult := fbDS402.fVelocity;

AssertEquals(Expected := fExpected,
             Actual := fResult,
             Message := 'Value is not correct');	 
TEST_FINISHED();
END_METHOD

METHOD TestSpeedModeEncoder : BOOL
VAR_INPUT
	sName 				: T_MaxString;
	nTarget				: DINT;
	fEncoderNumerator 	: REAL;
	fEncoderDenominator : REAL;	
	nExpected 			: DINT;
END_VAR

VAR
	fbDS402 			: FB_DS402;	
	nResult 			: DINT;
END_VAR
TEST(sName);

fbDS402.stConfig.eControlMode := E_ControlMode.Speed;
fbDS402.stConfig.fEncoderNumerator := fEncoderNumerator;
fbDS402.stConfig.fEncoderDenominator := fEncoderDenominator;
fbDS402.stConfig.fReferenceVelocity := 2000;

fbDS402.bSTO := TRUE;
EnableSequence(fbDS402);

fbDS402.nTargetValue := nTarget;

fbDS402();
nResult := fbDS402.nPosition;

AssertEquals(Expected := nExpected,
             Actual := nResult,
             Message := 'Value is not correct');	 
TEST_FINISHED();
END_METHOD

METHOD TestSpeedModeLinkOutput : BOOL
VAR_INPUT
	sName 				: T_MaxString;
	nTarget				: DINT;
	eLinkControlMode 	: E_ControlMode;
	fLinkOutputFactor	: REAL;	
	fExpected 			: REAL;
END_VAR

VAR
	fbDS402 			: FB_DS402;	
	fResult 			: REAL;
END_VAR
TEST(sName);

fbDS402.stConfig.eControlMode := E_ControlMode.Speed;
fbDS402.stConfig.fReferenceVelocity := 2000;
fbDS402.stConfig.eLinkControlMode := eLinkControlMode;
fbDS402.stConfig.fLinkOutputFactor := fLinkOutputFactor;

fbDS402.bSTO := TRUE;
EnableSequence(fbDS402);

fbDS402.nTargetValue := nTarget;

fbDS402();

fResult := fbDS402.GetLinkControlData();

AssertEquals(Expected := fExpected,
             Actual := fResult,
             Message := 'Value is not correct');	 
TEST_FINISHED();
END_METHOD

METHOD TestSpeedModeModulo : BOOL
VAR_INPUT
	sName 				: T_MaxString;
	nTarget				: DINT;
	fEncoderModulo	 	: REAL;	
	fExpected 			: REAL;
END_VAR

VAR
	fbDS402 			: FB_DS402;	
	fResult 			: REAL;
	nCycleCount 		: INT;
END_VAR
TEST(sName);

fbDS402.stConfig.eControlMode := E_ControlMode.Speed;
fbDS402.stConfig.fReferenceVelocity := 2000;
fbDS402.stConfig.fEncoderModulo := fEncoderModulo;

fbDS402.bSTO := TRUE;
EnableSequence(fbDS402);

fbDS402.nTargetValue := nTarget;

FOR nCycleCount := 1 TO 10 DO
    fbDS402();
END_FOR

fResult := fbDS402.fPosition;

AssertEquals(Expected := fExpected,
             Actual := fResult,
             Message := 'Value is not correct');	 
TEST_FINISHED();
END_METHOD

METHOD TestSpeedModeOffset : BOOL
VAR_INPUT
	sName 				: T_MaxString;
	nTarget				: DINT;
	fPositionOffset	 	: REAL;	
	fExpected 			: REAL;
END_VAR

VAR
	fbDS402 			: FB_DS402;	
	fResult 			: REAL;
END_VAR
TEST(sName);

fbDS402.stConfig.eControlMode := E_ControlMode.Speed;
fbDS402.stConfig.fReferenceVelocity := 2000;
fbDS402.stConfig.fPositionOffset := fPositionOffset;

fbDS402.bSTO := TRUE;
EnableSequence(fbDS402);

fbDS402.nTargetValue := nTarget;

fbDS402();

fResult := fbDS402.fPosition;

AssertEquals(Expected := fExpected,
             Actual := fResult,
             Message := 'Value is not correct');	 
TEST_FINISHED();
END_METHOD

END_FUNCTION_BLOCK

// Tests/Drives/FB_DS402FSM_Test
FUNCTION_BLOCK FB_DS402FSM_Test EXTENDS TcUnit.FB_TestSuite

TestState_S0();
TestState_S1();
TestState_S2();
TestState_S3();
TestState_S4();
TestState_S5();
TestState_S6();
TestState_S7();
TestEnableSequence();

METHOD GetDisableCommand : ST_DS402_6040h_ControlWord
GetDisableCommand.b0_SwitchOn := TRUE;
GetDisableCommand.b1_EnableVoltage := TRUE;
GetDisableCommand.b2_QuickStop := TRUE;
GetDisableCommand.b3_EnableOperation := FALSE;
GetDisableCommand.b7_FaultReset := FALSE;
END_METHOD

METHOD GetDisableVoltageCommand : ST_DS402_6040h_ControlWord
GetDisableVoltageCommand.b1_EnableVoltage := FALSE;
GetDisableVoltageCommand.b7_FaultReset := FALSE;
END_METHOD

METHOD GetEnableCommand : ST_DS402_6040h_ControlWord
GetEnableCommand.b0_SwitchOn := TRUE;
GetEnableCommand.b1_EnableVoltage := TRUE;
GetEnableCommand.b2_QuickStop := TRUE;
GetEnableCommand.b3_EnableOperation := TRUE;
GetEnableCommand.b7_FaultReset := FALSE;
END_METHOD

METHOD GetQuickStopCommand : ST_DS402_6040h_ControlWord
GetQuickStopCommand.b2_QuickStop := FALSE;
GetQuickStopCommand.b7_FaultReset := FALSE;
END_METHOD

METHOD GetShotdownCommand : ST_DS402_6040h_ControlWord
GetShotdownCommand.b0_SwitchOn := FALSE;
GetShotdownCommand.b1_EnableVoltage := TRUE;
GetShotdownCommand.b2_QuickStop := TRUE;
GetShotdownCommand.b7_FaultReset := FALSE;
END_METHOD

METHOD GetSwitchOnCommand : ST_DS402_6040h_ControlWord
GetSwitchOnCommand.b0_SwitchOn := TRUE;
GetSwitchOnCommand.b1_EnableVoltage := TRUE;
GetSwitchOnCommand.b2_QuickStop := TRUE;
GetSwitchOnCommand.b7_FaultReset := FALSE;
END_METHOD

METHOD TestEnableSequence : BOOL
VAR
	fbDS402 			: FB_DS402FSM;
	stExpectedStatus 	: ST_DS402_6041h_StatusWord; 
	nMask 				: WORD;
	nResult 			: WORD;
	bResult 			: BOOL;
	nActualState		: INT;
	nExpectedState		: INT;
END_VAR
TEST('Enable S1');

fbDS402();
nExpectedState := E_DS402State.S1_SwitchOnDisabled;
nActualState := fbDS402.eState;

AssertEquals(Expected := nExpectedState,
             Actual := nActualState,
             Message := 'State is not correct');	 
TEST_FINISHED();

TEST('Enable S2');
fbDS402.stControl.b1_EnableVoltage := TRUE;
fbDS402.stControl.b2_QuickStop := TRUE;

fbDS402();
nExpectedState := E_DS402State.S2_ReadyToSwitchOn;
nActualState := fbDS402.eState;

AssertEquals(Expected := nExpectedState,
             Actual := nActualState,
             Message := 'State is not correct');	 
TEST_FINISHED();

TEST('Enable S3');
fbDS402.stControl.b0_SwitchOn := TRUE;

fbDS402();
nExpectedState := E_DS402State.S3_SwitchedOn;
nActualState := fbDS402.eState;

AssertEquals(Expected := nExpectedState,
             Actual := nActualState,
             Message := 'State is not correct');	 
TEST_FINISHED();

TEST('Enable S4');
fbDS402.stControl.b3_EnableOperation := TRUE;

fbDS402();
nExpectedState := E_DS402State.S4_OperationEnabled;
nActualState := fbDS402.eState;

AssertEquals(Expected := nExpectedState,
             Actual := nActualState,
             Message := 'State is not correct');	 
TEST_FINISHED();

TEST('Disable S4');
fbDS402.stControl.b3_EnableOperation := FALSE;

fbDS402();
nExpectedState := E_DS402State.S3_SwitchedOn;
nActualState := fbDS402.eState;

AssertEquals(Expected := nExpectedState,
             Actual := nActualState,
             Message := 'State is not correct');	 
TEST_FINISHED();

TEST('Disable S3');
fbDS402.stControl.b0_SwitchOn := FALSE;

fbDS402();
nExpectedState := E_DS402State.S2_ReadyToSwitchOn;
nActualState := fbDS402.eState;

AssertEquals(Expected := nExpectedState,
             Actual := nActualState,
             Message := 'State is not correct');	 
TEST_FINISHED();

TEST('Disable S2');
fbDS402.stControl.b1_EnableVoltage := FALSE;
fbDS402.stControl.b2_QuickStop := FALSE;

fbDS402();
nExpectedState := E_DS402State.S1_SwitchOnDisabled;
nActualState := fbDS402.eState;

AssertEquals(Expected := nExpectedState,
             Actual := nActualState,
             Message := 'State is not correct');	 
TEST_FINISHED();
END_METHOD

METHOD TestState_S0 : BOOL
VAR
	fbDS402 			: FB_DS402FSM;
	stExpectedStatus 	: ST_DS402_6041h_StatusWord; 
	nMask 				: WORD;
	nResult 			: WORD;
	bResult 			: BOOL;
	nActualState		: INT;
	nExpectedState		: INT;
END_VAR
TEST('Set State S0');
fbDS402.eState := E_DS402State.S0_NotReadyToSwitchOn;
fbDS402();

stExpectedStatus.b0_ReadyToSwitchOn 		:= FALSE;
stExpectedStatus.b1_SwitchedOn 				:= FALSE;
stExpectedStatus.b2_OperationEnabled		:= FALSE;
stExpectedStatus.b3_Fault					:= FALSE;
stExpectedStatus.b4_VoltageEnabled			:= FALSE;
stExpectedStatus.b6_SwitchOnDisabled 		:= FALSE;

MEMCPY(ADR(nMask), ADR(stExpectedStatus), 2);
nResult := (2#01011111 AND fbDS402.nStatus);

AssertEquals(Expected := nMask,
             Actual := nResult,
             Message := 'Value is not correct');	 
TEST_FINISHED();

TEST('Transition S0>S1');
fbDS402.eState := E_DS402State.S0_NotReadyToSwitchOn;
fbDS402();
fbDS402();

nExpectedState := E_DS402State.S1_SwitchOnDisabled;
nActualState := fbDS402.eState;


AssertEquals(Expected := nExpectedState,
             Actual := nActualState,
             Message := 'State is not correct');	 
TEST_FINISHED();
END_METHOD

METHOD TestState_S1 : BOOL
VAR
	fbDS402 			: FB_DS402FSM;
	stExpectedStatus 	: ST_DS402_6041h_StatusWord; 
	nMask 				: WORD;
	nResult 			: WORD;
	bResult 			: BOOL;
	nActualState		: INT;
	nExpectedState		: INT;
END_VAR
TEST('Set State S1');
fbDS402.eState := E_DS402State.S1_SwitchOnDisabled;
fbDS402();

stExpectedStatus.b0_ReadyToSwitchOn 		:= FALSE;
stExpectedStatus.b1_SwitchedOn 				:= FALSE;
stExpectedStatus.b2_OperationEnabled		:= FALSE;
stExpectedStatus.b3_Fault					:= FALSE;
stExpectedStatus.b4_VoltageEnabled			:= FALSE;
stExpectedStatus.b6_SwitchOnDisabled 		:= TRUE;

MEMCPY(ADR(nMask), ADR(stExpectedStatus), 2);
nResult := (2#01011111 AND fbDS402.nStatus);

AssertEquals(Expected := nMask,
             Actual := nResult,
             Message := 'Value is not correct');	 
TEST_FINISHED();

TEST('Transition S1>S2');
fbDS402.eState := E_DS402State.S1_SwitchOnDisabled;
fbDS402.stControl := GetShotdownCommand();
fbDS402();

nExpectedState := E_DS402State.S2_ReadyToSwitchOn;
nActualState := fbDS402.eState;


AssertEquals(Expected := nExpectedState,
             Actual := nActualState,
             Message := 'State is not correct');	 
TEST_FINISHED();
END_METHOD

METHOD TestState_S2 : BOOL
VAR
	fbDS402 			: FB_DS402FSM;
	stExpectedStatus 	: ST_DS402_6041h_StatusWord; 
	nMask 				: WORD;
	nResult 			: WORD;
	bResult 			: BOOL;
	nActualState		: INT;
	nExpectedState		: INT;
END_VAR
TEST('Set State S2');
fbDS402.eState := E_DS402State.S2_ReadyToSwitchOn;
fbDS402();

stExpectedStatus.b0_ReadyToSwitchOn 		:= TRUE;
stExpectedStatus.b1_SwitchedOn 				:= FALSE;
stExpectedStatus.b2_OperationEnabled		:= FALSE;
stExpectedStatus.b3_Fault					:= FALSE;
stExpectedStatus.b4_VoltageEnabled			:= TRUE;
stExpectedStatus.b5_QuickStop 				:= TRUE; 
stExpectedStatus.b6_SwitchOnDisabled 		:= FALSE;

MEMCPY(ADR(nMask), ADR(stExpectedStatus), 2);
nResult := (2#01111111 AND fbDS402.nStatus);

AssertEquals(Expected := nMask,
             Actual := nResult,
             Message := 'Value is not correct');	 
TEST_FINISHED();

TEST('Transition S2>S6');
fbDS402.eState := E_DS402State.S2_ReadyToSwitchOn;
fbDS402.bError := TRUE;
fbDS402();
fbDS402.bError := FALSE;

nExpectedState := E_DS402State.S6_FaultReactionActive;
nActualState := fbDS402.eState;

AssertEquals(Expected := nExpectedState,
             Actual := nActualState,
             Message := 'State is not correct');	 
TEST_FINISHED();

TEST('Transition S2>S1_1');
fbDS402.eState := E_DS402State.S2_ReadyToSwitchOn;
fbDS402.stControl := GetDisableVoltageCommand();
fbDS402();

nExpectedState := E_DS402State.S1_SwitchOnDisabled;
nActualState := fbDS402.eState;

AssertEquals(Expected := nExpectedState,
             Actual := nActualState,
             Message := 'State is not correct');	 
TEST_FINISHED();

TEST('Transition S2>S1_2');
fbDS402.eState := E_DS402State.S2_ReadyToSwitchOn;
fbDS402.stControl := GetQuickStopCommand();
fbDS402.stControl.b1_EnableVoltage := TRUE;
fbDS402();

nExpectedState := E_DS402State.S1_SwitchOnDisabled;
nActualState := fbDS402.eState;

AssertEquals(Expected := nExpectedState,
             Actual := nActualState,
             Message := 'State is not correct');	 
TEST_FINISHED();

TEST('Transition S2>S3');
fbDS402.eState := E_DS402State.S2_ReadyToSwitchOn;
fbDS402.stControl := GetSwitchOnCommand();
fbDS402();

nExpectedState := E_DS402State.S3_SwitchedOn;
nActualState := fbDS402.eState;

AssertEquals(Expected := nExpectedState,
             Actual := nActualState,
             Message := 'State is not correct');	 
TEST_FINISHED();
END_METHOD

METHOD TestState_S3 : BOOL
VAR
	fbDS402 			: FB_DS402FSM;
	stExpectedStatus 	: ST_DS402_6041h_StatusWord; 
	nMask 				: WORD;
	nResult 			: WORD;
	bResult 			: BOOL;
	nActualState		: INT;
	nExpectedState		: INT;
END_VAR
TEST('Set State S3');
fbDS402.eState := E_DS402State.S3_SwitchedOn;
fbDS402();

stExpectedStatus.b0_ReadyToSwitchOn 		:= TRUE;
stExpectedStatus.b1_SwitchedOn 				:= TRUE;
stExpectedStatus.b2_OperationEnabled		:= FALSE;
stExpectedStatus.b3_Fault					:= FALSE;
stExpectedStatus.b5_QuickStop 				:= TRUE; 
stExpectedStatus.b6_SwitchOnDisabled 		:= FALSE;

MEMCPY(ADR(nMask), ADR(stExpectedStatus), 2);
nResult := (2#01101111 AND fbDS402.nStatus);

AssertEquals(Expected := nMask,
             Actual := nResult,
             Message := 'Value is not correct');	 
TEST_FINISHED();

TEST('Transition S3>S6');
fbDS402.eState := E_DS402State.S3_SwitchedOn;
fbDS402.bError := TRUE;
fbDS402();
fbDS402.bError := FALSE;

nExpectedState := E_DS402State.S6_FaultReactionActive;
nActualState := fbDS402.eState;

AssertEquals(Expected := nExpectedState,
             Actual := nActualState,
             Message := 'State is not correct');	 
TEST_FINISHED();

TEST('Transition S3>S1_1');
fbDS402.eState := E_DS402State.S3_SwitchedOn;
fbDS402.stControl := GetDisableVoltageCommand();
fbDS402();

nExpectedState := E_DS402State.S1_SwitchOnDisabled;
nActualState := fbDS402.eState;

